C07362=1109.308,78.627,-56.858,-179.889,7.756,149.437
C07363=1109.304,78.877,-56.876,-179.889,7.759,149.437
C07364=1109.299,79.126,-56.895,-179.887,7.763,149.438
C07365=1109.295,79.375,-56.913,-179.887,7.767,149.438
C07366=1109.289,79.625,-56.931,-179.885,7.770,149.439
C07367=1109.285,79.874,-56.949,-179.885,7.774,149.440
C07368=1109.280,80.124,-56.967,-179.883,7.778,149.440
C07369=1109.275,80.372,-56.986,-179.883,7.781,149.441
C07370=1109.270,80.621,-57.004,-179.881,7.785,149.441
C07371=1109.266,80.871,-57.022,-179.880,7.790,149.442
C07372=1109.260,81.121,-57.041,-179.879,7.793,149.442
C07373=1109.255,81.370,-57.059,-179.878,7.797,149.443
C07374=1109.251,81.618,-57.078,-179.877,7.800,149.443
C07375=1109.246,81.868,-57.096,-179.876,7.804,149.444
C07376=1109.241,82.118,-57.115,-179.875,7.807,149.444
C07377=1109.236,82.367,-57.133,-179.874,7.812,149.445
C07378=1109.231,82.615,-57.151,-179.873,7.815,149.445
C07379=1109.227,82.865,-57.170,-179.872,7.819,149.446
C07380=1109.222,83.115,-57.188,-179.870,7.823,149.446
C07381=1109.217,83.363,-57.207,-179.869,7.827,149.447
C07382=1109.212,83.613,-57.225,-179.868,7.830,149.448
C07383=1109.207,83.862,-57.243,-179.867,7.834,149.448
C07384=1109.202,84.111,-57.263,-179.866,7.838,149.449
C07385=1109.198,84.361,-57.281,-179.865,7.842,149.449
C07386=1109.193,84.610,-57.299,-179.864,7.845,149.450
C07387=1109.188,84.859,-57.318,-179.863,7.849,149.450
C07388=1109.183,85.109,-57.337,-179.862,7.853,149.451
C07389=1109.179,85.358,-57.355,-179.860,7.856,149.451
C07390=1109.174,85.607,-57.373,-179.859,7.861,149.452
C07391=1109.169,85.857,-57.392,-179.858,7.864,149.452
C07392=1109.164,86.106,-57.411,-179.857,7.868,149.453
C07393=1109.159,86.355,-57.429,-179.855,7.872,149.453
C07394=1109.154,86.604,-57.448,-179.855,7.876,149.454
C07395=1109.149,86.854,-57.466,-179.853,7.879,149.454
C07396=1109.145,87.102,-57.485,-179.852,7.883,149.455
C07397=1109.140,87.352,-57.504,-179.851,7.887,149.456
C07398=1109.135,87.601,-57.523,-179.849,7.891,149.456
C07399=1109.130,87.851,-57.542,-179.848,7.895,149.456
C07400=1109.126,88.100,-57.560,-179.847,7.898,149.457
C07401=1109.121,88.349,-57.578,-179.846,7.902,149.458
C07402=1109.116,88.598,-57.598,-179.844,7.906,149.458
C07403=1109.111,88.847,-57.616,-179.844,7.909,149.459
C07404=1109.106,89.096,-57.635,-179.842,7.913,149.459
C07405=1109.101,89.346,-57.654,-179.840,7.917,149.459
C07406=1109.097,89.595,-57.672,-179.839,7.921,149.460
C07407=1109.092,89.845,-57.691,-179.838,7.925,149.461
C07408=1109.087,90.094,-57.710,-179.837,7.928,149.461
C07409=1109.082,90.343,-57.730,-179.836,7.933,149.462
C07410=1109.077,90.592,-57.748,-179.835,7.936,149.462
C07411=1109.074,90.806,-57.764,-179.833,7.940,149.462
C07412=1109.069,91.019,-57.781,-179.832,7.943,149.463
C07413=1109.065,91.234,-57.797,-179.831,7.946,149.463
C07414=1109.060,91.447,-57.813,-179.830,7.949,149.464
C07415=1109.057,91.661,-57.829,-179.829,7.953,149.464
C07416=1109.053,91.875,-57.845,-179.827,7.956,149.464
C07417=1109.049,92.088,-57.861,-179.826,7.959,149.465
C07418=1109.044,92.302,-57.878,-179.825,7.962,149.465
C07419=1109.039,92.551,-57.896,-179.824,7.966,149.466
C07420=1109.035,92.801,-57.916,-179.822,7.970,149.466
C07421=1109.030,93.050,-57.934,-179.821,7.974,149.467
C07422=1109.025,93.299,-57.954,-179.820,7.977,149.467
C07423=1109.020,93.548,-57.972,-179.818,7.981,149.468
C07424=1109.016,93.798,-57.992,-179.817,7.985,149.468
C07425=1109.011,94.046,-58.010,-179.815,7.989,149.469
C07426=1109.006,94.296,-58.030,-179.815,7.992,149.469
C07427=1109.001,94.546,-58.048,-179.813,7.996,149.470
C07428=1108.997,94.795,-58.068,-179.811,8.000,149.470
C07429=1108.991,95.044,-58.087,-179.810,8.004,149.471
C07430=1108.987,95.293,-58.106,-179.808,8.008,149.471
C07431=1108.982,95.542,-58.125,-179.807,8.012,149.471
C07432=1108.977,95.792,-58.144,-179.806,8.015,149.472
C07433=1108.972,96.041,-58.163,-179.804,8.019,149.472
C07434=1108.967,96.290,-58.182,-179.802,8.022,149.473
C07435=1108.963,96.539,-58.202,-179.801,8.026,149.473
C07436=1108.958,96.788,-58.221,-179.799,8.030,149.474
C07437=1108.953,97.038,-58.240,-179.798,8.033,149.474
C07438=1108.949,97.286,-58.259,-179.797,8.037,149.474
C07439=1108.944,97.537,-58.278,-179.795,8.041,149.475
C07440=1108.938,97.785,-58.297,-179.793,8.045,149.475
C07441=1108.934,98.035,-58.316,-179.792,8.049,149.476
C07442=1108.929,98.284,-58.336,-179.790,8.053,149.476
C07443=1108.924,98.533,-58.355,-179.789,8.057,149.477
C07444=1108.920,98.782,-58.374,-179.788,8.060,149.477
C07445=1108.915,99.031,-58.394,-179.786,8.064,149.477
C07446=1108.910,99.281,-58.413,-179.784,8.068,149.478
C07447=1108.905,99.530,-58.433,-179.783,8.071,149.478
C07448=1108.901,99.779,-58.452,-179.781,8.075,149.479
C07449=1108.896,100.028,-58.471,-179.780,8.079,149.479
C07450=1108.891,100.277,-58.491,-179.778,8.083,149.480
C07451=1108.886,100.527,-58.510,-179.776,8.087,149.480
C07452=1108.881,100.775,-58.529,-179.774,8.091,149.480
C07453=1108.877,101.025,-58.549,-179.773,8.094,149.481
C07454=1108.872,101.275,-58.568,-179.772,8.098,149.481
C07455=1108.867,101.523,-58.588,-179.770,8.101,149.482
C07456=1108.863,101.772,-58.607,-179.769,8.105,149.482
C07457=1108.858,102.022,-58.627,-179.766,8.109,149.482
C07458=1108.853,102.271,-58.646,-179.765,8.113,149.483
C07459=1108.848,102.520,-58.666,-179.763,8.117,149.483
C07460=1108.843,102.770,-58.686,-179.762,8.120,149.484
C07461=1108.839,103.018,-58.704,-179.760,8.124,149.484
C07462=1108.834,103.268,-58.724,-179.758,8.128,149.484
C07463=1108.829,103.517,-58.744,-179.756,8.132,149.485
C07464=1108.824,103.766,-58.764,-179.755,8.134,149.485
C07465=1108.819,104.015,-58.783,-179.753,8.138,149.485
C07466=1108.815,104.265,-58.803,-179.752,8.142,149.486
C07467=1108.811,104.478,-58.820,-179.750,8.146,149.486
C07468=1108.806,104.692,-58.836,-179.749,8.149,149.486
C07469=1108.802,104.905,-58.853,-179.747,8.152,149.487
C07470=1108.798,105.119,-58.870,-179.745,8.155,149.487
C07471=1108.795,105.333,-58.887,-179.744,8.158,149.487
C07472=1108.790,105.547,-58.904,-179.742,8.162,149.488
C07473=1108.786,105.760,-58.920,-179.741,8.164,149.488
C07474=1108.782,105.974,-58.938,-179.740,8.167,149.488
C07475=1108.777,106.223,-58.957,-179.738,8.171,149.488
C07476=1108.773,106.472,-58.978,-179.736,8.175,149.489
C07477=1108.768,106.722,-58.997,-179.734,8.178,149.489
C07478=1108.763,106.971,-59.017,-179.732,8.182,149.490
C07479=1108.758,107.220,-59.037,-179.730,8.186,149.490
C07480=1108.753,107.469,-59.057,-179.729,8.190,149.490
C07481=1108.749,107.719,-59.076,-179.727,8.193,149.490
C07482=1108.744,107.967,-59.096,-179.725,8.197,149.491
C07483=1108.740,108.216,-59.116,-179.723,8.201,149.491
C07484=1108.735,108.466,-59.135,-179.721,8.204,149.491
C07485=1108.730,108.715,-59.156,-179.719,8.208,149.492
C07486=1108.725,108.965,-59.176,-179.717,8.211,149.492
C07487=1108.720,109.213,-59.196,-179.716,8.215,149.492
C07488=1108.715,109.462,-59.215,-179.714,8.219,149.493
C07489=1108.711,109.711,-59.236,-179.712,8.222,149.493
C07490=1108.706,109.961,-59.255,-179.710,8.226,149.493
C07491=1108.701,110.210,-59.276,-179.708,8.230,149.494
C07492=1108.696,110.459,-59.295,-179.706,8.233,149.494
C07493=1108.692,110.708,-59.316,-179.704,8.237,149.494
C07494=1108.687,110.957,-59.335,-179.702,8.241,149.494
C07495=1108.683,111.206,-59.356,-179.700,8.244,149.495
C07496=1108.678,111.456,-59.375,-179.699,8.247,149.495
C07497=1108.673,111.704,-59.395,-179.697,8.251,149.495
C07498=1108.668,111.954,-59.415,-179.695,8.254,149.496
C07499=1108.663,112.203,-59.436,-179.693,8.258,149.496
C07500=1108.658,112.452,-59.455,-179.692,8.261,149.496
C07501=1108.654,112.701,-59.476,-179.690,8.264,149.496
C07502=1108.649,112.950,-59.496,-179.688,8.268,149.497
C07503=1108.644,113.200,-59.516,-179.686,8.272,149.497
C07504=1108.640,113.449,-59.536,-179.685,8.274,149.497
C07505=1108.635,113.697,-59.556,-179.683,8.278,149.498
C07506=1108.630,113.947,-59.577,-179.681,8.282,149.498
C07507=1108.625,114.196,-59.597,-179.680,8.284,149.498
C07508=1108.621,114.445,-59.617,-179.678,8.288,149.499
C07509=1108.616,114.694,-59.637,-179.676,8.292,149.499
C07510=1108.611,114.943,-59.657,-179.674,8.295,149.499
C07511=1108.606,115.193,-59.678,-179.673,8.298,149.500
C07512=1108.602,115.442,-59.698,-179.671,8.302,149.500
C07513=1108.597,115.691,-59.718,-179.669,8.305,149.500
C07514=1108.593,115.940,-59.739,-179.668,8.309,149.500
C07515=1108.587,116.189,-59.759,-179.666,8.312,149.501
C07516=1108.582,116.438,-59.779,-179.664,8.316,149.501
C07517=1108.578,116.687,-59.799,-179.662,8.319,149.501
C07518=1108.573,116.936,-59.820,-179.661,8.322,149.502
C07519=1108.568,117.185,-59.841,-179.659,8.326,149.502
C07520=1108.563,117.435,-59.860,-179.657,8.329,149.502
C07521=1108.559,117.684,-59.881,-179.656,8.332,149.502
C07522=1108.554,117.933,-59.901,-179.654,8.336,149.503
C07523=1108.550,118.147,-59.918,-179.652,8.338,149.503
C07524=1108.546,118.360,-59.937,-179.651,8.341,149.503
C07525=1108.542,118.574,-59.954,-179.649,8.345,149.503
C07526=1108.538,118.787,-59.971,-179.647,8.347,149.504
C07527=1108.534,119.001,-59.990,-179.646,8.350,149.504
C07528=1108.530,119.214,-60.007,-179.645,8.353,149.504
C07529=1108.526,119.428,-60.024,-179.643,8.356,149.504
C07530=1108.522,119.641,-60.042,-179.642,8.359,149.505
C07531=1108.517,119.891,-60.062,-179.640,8.362,149.505
C07532=1108.512,120.140,-60.082,-179.638,8.366,149.505
C07533=1108.508,120.389,-60.103,-179.637,8.369,149.506
C07534=1108.503,120.638,-60.124,-179.635,8.372,149.506
C07535=1108.498,120.887,-60.144,-179.633,8.376,149.506
C07536=1108.494,121.136,-60.165,-179.631,8.378,149.506
C07537=1108.489,121.385,-60.186,-179.630,8.382,149.507
C07538=1108.485,121.635,-60.206,-179.628,8.386,149.507
C07539=1108.480,121.884,-60.227,-179.625,8.389,149.507
C07540=1108.475,122.133,-60.248,-179.624,8.392,149.507
C07541=1108.471,122.382,-60.268,-179.622,8.396,149.508
C07542=1108.465,122.631,-60.289,-179.620,8.399,149.508
C07543=1108.461,122.880,-60.309,-179.619,8.402,149.508
C07544=1108.456,123.129,-60.330,-179.617,8.406,149.508
C07545=1108.451,123.378,-60.351,-179.615,8.410,149.509
C07546=1108.447,123.627,-60.372,-179.614,8.412,149.509
C07547=1108.442,123.876,-60.393,-179.612,8.416,149.509
C07548=1108.437,124.125,-60.414,-179.610,8.419,149.510
C07549=1108.433,124.374,-60.434,-179.609,8.422,149.510
C07550=1108.428,124.623,-60.454,-179.607,8.426,149.510
C07551=1108.424,124.873,-60.476,-179.605,8.429,149.511
C07552=1108.419,125.122,-60.496,-179.603,8.432,149.511
C07553=1108.414,125.371,-60.517,-179.601,8.436,149.511
C07554=1108.410,125.620,-60.538,-179.599,8.439,149.511
C07555=1108.405,125.869,-60.559,-179.598,8.442,149.512
C07556=1108.399,126.118,-60.580,-179.596,8.446,149.512
C07557=1108.395,126.367,-60.600,-179.594,8.449,149.512
C07558=1108.390,126.616,-60.621,-179.592,8.453,149.513
C07559=1108.386,126.865,-60.643,-179.591,8.456,149.513
C07560=1108.381,127.115,-60.664,-179.589,8.459,149.513
C07561=1108.377,127.364,-60.684,-179.587,8.463,149.513
C07562=1108.371,127.613,-60.705,-179.586,8.466,149.514
C07563=1108.367,127.861,-60.726,-179.584,8.469,149.514
C07564=1108.362,128.110,-60.747,-179.582,8.473,149.514
C07565=1108.357,128.360,-60.768,-179.580,8.475,149.514
C07566=1108.353,128.609,-60.789,-179.578,8.479,149.515
C07567=1108.348,128.858,-60.811,-179.576,8.483,149.515
C07568=1108.343,129.107,-60.832,-179.575,8.486,149.515
C07569=1108.339,129.356,-60.852,-179.573,8.489,149.515
C07570=1108.334,129.605,-60.874,-179.571,8.493,149.516
C07571=1108.330,129.854,-60.894,-179.570,8.496,149.516
C07572=1108.325,130.103,-60.916,-179.568,8.499,149.516
C07573=1108.320,130.352,-60.937,-179.566,8.503,149.517
C07574=1108.316,130.601,-60.957,-179.565,8.506,149.517
C07575=1108.311,130.850,-60.979,-179.563,8.509,149.517
C07576=1108.306,131.100,-61.000,-179.561,8.513,149.518
C07577=1108.301,131.349,-61.022,-179.559,8.515,149.518
C07578=1108.297,131.598,-61.043,-179.557,8.519,149.518
C07579=1108.293,131.811,-61.061,-179.556,8.522,149.518
C07580=1108.288,132.024,-61.079,-179.555,8.525,149.519
C07581=1108.284,132.239,-61.097,-179.552,8.528,149.519
C07582=1108.281,132.452,-61.115,-179.551,8.531,149.519
C07583=1108.277,132.665,-61.133,-179.550,8.534,149.519
C07584=1108.273,132.878,-61.152,-179.548,8.536,149.520
C07585=1108.268,133.092,-61.170,-179.547,8.539,149.520
C07586=1108.265,133.305,-61.189,-179.545,8.542,149.520
C07587=1108.259,133.555,-61.210,-179.544,8.546,149.520
C07588=1108.255,133.803,-61.231,-179.542,8.549,149.521
C07589=1108.251,134.053,-61.252,-179.540,8.552,149.521
C07590=1108.246,134.302,-61.274,-179.539,8.556,149.521
C07591=1108.241,134.551,-61.295,-179.536,8.559,149.522
C07592=1108.237,134.799,-61.316,-179.534,8.563,149.522
C07593=1108.232,135.049,-61.338,-179.533,8.565,149.522
C07594=1108.227,135.298,-61.359,-179.531,8.569,149.522
C07595=1108.222,135.546,-61.381,-179.529,8.573,149.523
C07596=1108.218,135.796,-61.402,-179.528,8.576,149.523
C07597=1108.214,136.045,-61.423,-179.526,8.579,149.523
C07598=1108.209,136.293,-61.445,-179.524,8.583,149.524
C07599=1108.204,136.543,-61.466,-179.523,8.586,149.524
C07600=1108.199,136.792,-61.488,-179.521,8.590,149.524
C07601=1108.194,137.041,-61.509,-179.519,8.593,149.525
C07602=1108.190,137.291,-61.531,-179.517,8.596,149.525
C07603=1108.185,137.539,-61.552,-179.515,8.599,149.525
C07604=1108.181,137.788,-61.573,-179.514,8.603,149.525
C07605=1108.176,138.038,-61.595,-179.512,8.607,149.526
C07606=1108.171,138.286,-61.616,-179.510,8.609,149.526
C07607=1108.166,138.535,-61.638,-179.509,8.613,149.526
C07608=1108.162,138.784,-61.660,-179.507,8.617,149.527
C07609=1108.157,139.033,-61.681,-179.505,8.621,149.527
C07610=1108.152,139.282,-61.703,-179.503,8.623,149.527
C07611=1108.148,139.531,-61.725,-179.501,8.627,149.527
C07612=1108.143,139.780,-61.747,-179.500,8.631,149.528
C07613=1108.139,140.029,-61.769,-179.498,8.633,149.528
C07614=1108.134,140.279,-61.790,-179.496,8.637,149.528
C07615=1108.129,140.527,-61.811,-179.495,8.641,149.529
C07616=1108.124,140.777,-61.833,-179.493,8.644,149.529
C07617=1108.120,141.025,-61.854,-179.491,8.647,149.529
C07618=1108.116,141.274,-61.876,-179.489,8.651,149.530
C07619=1108.111,141.523,-61.898,-179.487,8.654,149.530
C07620=1108.107,141.772,-61.920,-179.486,8.657,149.530
C07621=1108.102,142.022,-61.941,-179.484,8.661,149.531
C07622=1108.097,142.270,-61.963,-179.482,8.664,149.531
C07623=1108.093,142.520,-61.985,-179.481,8.668,149.531
C07624=1108.088,142.768,-62.007,-179.479,8.671,149.532
C07625=1108.083,143.017,-62.029,-179.477,8.675,149.532
C07626=1108.078,143.266,-62.051,-179.475,8.678,149.532
C07627=1108.074,143.516,-62.073,-179.474,8.682,149.533
C07628=1108.069,143.764,-62.095,-179.472,8.685,149.533
C07629=1108.064,144.014,-62.117,-179.470,8.688,149.533
C07630=1108.060,144.262,-62.138,-179.469,8.692,149.534
C07631=1108.055,144.512,-62.160,-179.467,8.696,149.534
C07632=1108.050,144.760,-62.182,-179.466,8.699,149.534
C07633=1108.046,145.010,-62.204,-179.463,8.702,149.534
C07634=1108.041,145.258,-62.226,-179.462,8.706,149.535
C07635=1108.037,145.471,-62.245,-179.460,8.709,149.535
C07636=1108.034,145.685,-62.264,-179.458,8.712,149.535
C07637=1108.029,145.899,-62.282,-179.457,8.715,149.536
C07638=1108.026,146.112,-62.302,-179.455,8.718,149.536
C07639=1108.021,146.325,-62.320,-179.453,8.721,149.536
C07640=1108.017,146.538,-62.339,-179.452,8.724,149.537
C07641=1108.013,146.752,-62.358,-179.450,8.728,149.537
C07642=1108.010,146.965,-62.376,-179.449,8.730,149.537
C07643=1108.005,147.215,-62.398,-179.447,8.734,149.537
C07644=1108.000,147.463,-62.421,-179.445,8.737,149.537
C07645=1107.996,147.712,-62.444,-179.443,8.741,149.538
C07646=1107.991,147.961,-62.465,-179.441,8.745,149.538
C07647=1107.987,148.210,-62.487,-179.439,8.748,149.538
C07648=1107.982,148.460,-62.509,-179.437,8.751,149.539
C07649=1107.977,148.708,-62.532,-179.435,8.755,149.539
C07650=1107.973,148.957,-62.554,-179.433,8.758,149.539
C07651=1107.968,149.206,-62.576,-179.431,8.761,149.539
C07652=1107.964,149.455,-62.598,-179.429,8.765,149.540
C07653=1107.958,149.704,-62.620,-179.427,8.768,149.540
C07654=1107.954,149.953,-62.643,-179.425,8.772,149.540
C07655=1107.950,150.202,-62.665,-179.423,8.776,149.540
C07656=1107.945,150.451,-62.687,-179.422,8.779,149.541
C07657=1107.940,150.700,-62.709,-179.420,8.782,149.541
C07658=1107.935,150.948,-62.732,-179.418,8.785,149.541
C07659=1107.931,151.198,-62.754,-179.416,8.789,149.541
C07660=1107.926,151.447,-62.777,-179.413,8.792,149.542
C07661=1107.921,151.695,-62.799,-179.411,8.796,149.542
C07662=1107.917,151.945,-62.821,-179.409,8.799,149.542
C07663=1107.912,152.193,-62.844,-179.407,8.802,149.542
C07664=1107.908,152.443,-62.866,-179.405,8.805,149.542
C07665=1107.903,152.692,-62.888,-179.403,8.809,149.543
C07666=1107.898,152.940,-62.911,-179.401,8.812,149.543
C07667=1107.894,153.190,-62.933,-179.399,8.816,149.543
C07668=1107.890,153.438,-62.956,-179.397,8.819,149.543
C07669=1107.884,153.687,-62.978,-179.396,8.822,149.544
C07670=1107.880,153.937,-63.000,-179.393,8.825,149.544
C07671=1107.875,154.186,-63.024,-179.391,8.829,149.544
C07672=1107.870,154.434,-63.045,-179.389,8.832,149.544
C07673=1107.866,154.683,-63.068,-179.387,8.836,149.544
C07674=1107.861,154.933,-63.091,-179.385,8.838,149.545
C07675=1107.857,155.181,-63.113,-179.383,8.842,149.545
C07676=1107.852,155.430,-63.136,-179.381,8.845,149.545
C07677=1107.848,155.679,-63.159,-179.379,8.849,149.545
C07678=1107.843,155.928,-63.180,-179.377,8.852,149.545
C07679=1107.838,156.177,-63.204,-179.375,8.854,149.546
C07680=1107.834,156.425,-63.226,-179.373,8.858,149.546
C07681=1107.829,156.675,-63.249,-179.371,8.861,149.546
C07682=1107.825,156.923,-63.271,-179.368,8.865,149.546
C07683=1107.820,157.173,-63.294,-179.366,8.868,149.546
C07684=1107.816,157.421,-63.317,-179.365,8.871,149.547
C07685=1107.811,157.670,-63.340,-179.362,8.874,149.547
C07686=1107.806,157.919,-63.362,-179.360,8.877,149.547
C07687=1107.802,158.168,-63.385,-179.358,8.881,149.547
C07688=1107.798,158.417,-63.408,-179.356,8.883,149.547
C07689=1107.793,158.667,-63.431,-179.354,8.887,149.547
C07690=1107.788,158.915,-63.453,-179.352,8.890,149.548
C07691=1107.784,159.128,-63.473,-179.350,8.892,149.548
C07692=1107.780,159.342,-63.493,-179.349,8.895,149.548
C07693=1107.776,159.554,-63.512,-179.347,8.898,149.548
C07694=1107.772,159.768,-63.532,-179.345,8.901,149.548
C07695=1107.768,159.981,-63.551,-179.343,8.903,149.548
C07696=1107.764,160.194,-63.571,-179.341,8.906,149.548
C07697=1107.761,160.408,-63.590,-179.340,8.909,149.549
C07698=1107.757,160.621,-63.610,-179.338,8.911,149.549
C07699=1107.752,160.870,-63.633,-179.336,8.915,149.549
C07700=1107.748,161.119,-63.655,-179.334,8.918,149.549
C07701=1107.743,161.368,-63.678,-179.331,8.921,149.549
C07702=1107.738,161.617,-63.702,-179.330,8.924,149.549
C07703=1107.734,161.865,-63.724,-179.327,8.927,149.549
C07704=1107.729,162.114,-63.748,-179.325,8.930,149.549
C07705=1107.724,162.364,-63.770,-179.323,8.933,149.550
C07706=1107.720,162.612,-63.793,-179.321,8.936,149.550
C07707=1107.715,162.861,-63.816,-179.319,8.939,149.550
C07708=1107.711,163.110,-63.840,-179.317,8.943,149.550
C07709=1107.706,163.358,-63.862,-179.315,8.945,149.550
C07710=1107.701,163.608,-63.885,-179.313,8.949,149.550
C07711=1107.697,163.857,-63.909,-179.310,8.952,149.551
C07712=1107.693,164.105,-63.932,-179.309,8.955,149.551
C07713=1107.688,164.354,-63.955,-179.306,8.958,149.551
C07714=1107.683,164.603,-63.978,-179.304,8.961,149.551
C07715=1107.679,164.852,-64.001,-179.302,8.964,149.551
C07716=1107.675,165.101,-64.024,-179.300,8.967,149.551
C07717=1107.670,165.350,-64.048,-179.298,8.970,149.551
C07718=1107.665,165.598,-64.071,-179.295,8.973,149.551
C07719=1107.661,165.847,-64.094,-179.294,8.976,149.552
C07720=1107.656,166.096,-64.117,-179.291,8.979,149.552
C07721=1107.651,166.345,-64.140,-179.289,8.982,149.552
C07722=1107.647,166.594,-64.164,-179.287,8.985,149.552
C07723=1107.643,166.843,-64.186,-179.285,8.988,149.552
C07724=1107.638,167.092,-64.210,-179.283,8.991,149.552
C07725=1107.633,167.341,-64.233,-179.281,8.994,149.552
C07726=1107.629,167.590,-64.256,-179.279,8.997,149.552
C07727=1107.624,167.839,-64.280,-179.276,9.000,149.553
C07728=1107.619,168.088,-64.303,-179.275,9.003,149.553
C07729=1107.615,168.337,-64.326,-179.272,9.006,149.553
C07730=1107.611,168.586,-64.349,-179.270,9.009,149.553
C07731=1107.606,168.834,-64.373,-179.268,9.012,149.553
C07732=1107.601,169.083,-64.396,-179.266,9.015,149.553
C07733=1107.596,169.332,-64.420,-179.263,9.018,149.553
C07734=1107.591,169.581,-64.443,-179.262,9.021,149.553
C07735=1107.587,169.830,-64.466,-179.259,9.024,149.553
C07736=1107.583,170.078,-64.490,-179.257,9.027,149.554
C07737=1107.578,170.327,-64.513,-179.255,9.030,149.554
C07738=1107.574,170.576,-64.537,-179.253,9.033,149.554
C07739=1107.569,170.825,-64.560,-179.251,9.036,149.554
C07740=1107.565,171.073,-64.584,-179.249,9.039,149.554
C07741=1107.560,171.322,-64.607,-179.246,9.042,149.554
C07742=1107.555,171.571,-64.631,-179.244,9.045,149.554
C07743=1107.551,171.820,-64.654,-179.242,9.048,149.554
C07744=1107.546,172.069,-64.678,-179.240,9.051,149.554
C07745=1107.541,172.318,-64.702,-179.238,9.054,149.555
C07746=1107.537,172.568,-64.725,-179.236,9.057,149.555
C07747=1107.533,172.780,-64.745,-179.234,9.059,149.555
C07748=1107.530,172.993,-64.765,-179.232,9.062,149.555
C07749=1107.526,173.206,-64.786,-179.230,9.065,149.555
C07750=1107.522,173.420,-64.806,-179.228,9.067,149.555
C07751=1107.518,173.633,-64.827,-179.226,9.069,149.555
C07752=1107.514,173.845,-64.847,-179.225,9.072,149.555
C07753=1107.510,174.059,-64.867,-179.223,9.074,149.555
C07754=1107.507,174.272,-64.887,-179.221,9.077,149.555
C07755=1107.501,174.521,-64.911,-179.219,9.080,149.556
C07756=1107.497,174.770,-64.935,-179.216,9.083,149.556
C07757=1107.492,175.019,-64.959,-179.214,9.086,149.556
C07758=1107.488,175.268,-64.982,-179.212,9.089,149.556
C07759=1107.483,175.516,-65.006,-179.210,9.092,149.556
C07760=1107.479,175.766,-65.030,-179.208,9.095,149.556
C07761=1107.475,176.014,-65.054,-179.206,9.098,149.556
C07762=1107.470,176.263,-65.077,-179.203,9.101,149.556
C07763=1107.466,176.512,-65.101,-179.201,9.104,149.556
C07764=1107.461,176.761,-65.125,-179.199,9.107,149.557
C07765=1107.456,177.009,-65.149,-179.197,9.109,149.557
C07766=1107.452,177.258,-65.172,-179.195,9.113,149.557
C07767=1107.447,177.507,-65.196,-179.192,9.116,149.557
C07768=1107.444,177.756,-65.221,-179.191,9.118,149.557
C07769=1107.438,178.005,-65.244,-179.188,9.121,149.557
C07770=1107.434,178.253,-65.269,-179.186,9.125,149.557
C07771=1107.429,178.503,-65.292,-179.184,9.127,149.557
C07772=1107.425,178.751,-65.316,-179.182,9.130,149.557
C07773=1107.420,178.999,-65.340,-179.179,9.133,149.557
C07774=1107.416,179.249,-65.364,-179.178,9.136,149.558
C07775=1107.412,179.497,-65.388,-179.175,9.139,149.558
C07776=1107.407,179.746,-65.413,-179.173,9.142,149.558
C07777=1107.402,179.995,-65.436,-179.171,9.146,149.558
C07778=1107.398,180.244,-65.460,-179.169,9.148,149.558
C07779=1107.394,180.493,-65.484,-179.166,9.151,149.558
C07780=1107.389,180.742,-65.508,-179.164,9.154,149.558
C07781=1107.384,180.991,-65.532,-179.161,9.158,149.558
C07782=1107.379,181.239,-65.556,-179.159,9.160,149.558
C07783=1107.375,181.487,-65.581,-179.157,9.163,149.558
C07784=1107.371,181.737,-65.604,-179.155,9.166,149.558
C07785=1107.366,181.986,-65.629,-179.153,9.169,149.558
C07786=1107.361,182.234,-65.653,-179.150,9.172,149.559
C07787=1107.357,182.483,-65.677,-179.148,9.175,149.559
C07788=1107.353,182.732,-65.702,-179.146,9.177,149.559
C07789=1107.348,182.981,-65.726,-179.143,9.180,149.559
C07790=1107.343,183.229,-65.750,-179.141,9.184,149.559
C07791=1107.339,183.478,-65.774,-179.138,9.187,149.559
C07792=1107.335,183.727,-65.799,-179.136,9.189,149.559
C07793=1107.330,183.976,-65.823,-179.134,9.192,149.559
C07794=1107.326,184.224,-65.847,-179.131,9.195,149.559
C07795=1107.321,184.473,-65.871,-179.130,9.198,149.559
C07796=1107.317,184.723,-65.895,-179.127,9.201,149.559
C07797=1107.312,184.971,-65.919,-179.125,9.204,149.559
C07798=1107.307,185.220,-65.944,-179.123,9.206,149.559
C07799=1107.303,185.469,-65.968,-179.120,9.210,149.559
C07800=1107.299,185.717,-65.992,-179.119,9.212,149.559
C07801=1107.294,185.966,-66.017,-179.116,9.215,149.559
C07802=1107.289,186.214,-66.041,-179.114,9.218,149.559
C07803=1107.285,186.428,-66.062,-179.112,9.220,149.559
C07804=1107.282,186.641,-66.083,-179.110,9.223,149.559
C07805=1107.277,186.854,-66.104,-179.107,9.225,149.559
C07806=1107.274,187.066,-66.125,-179.106,9.227,149.559
C07807=1107.270,187.279,-66.146,-179.104,9.229,149.559
C07808=1107.266,187.493,-66.167,-179.102,9.232,149.559
C07809=1107.262,187.706,-66.188,-179.100,9.234,149.559
C07810=1107.258,187.919,-66.209,-179.097,9.237,149.560
C07811=1107.254,188.168,-66.234,-179.095,9.240,149.560
C07812=1107.249,188.417,-66.258,-179.093,9.243,149.560
C07813=1107.245,188.666,-66.283,-179.091,9.245,149.560
C07814=1107.240,188.914,-66.307,-179.089,9.248,149.560
C07815=1107.236,189.162,-66.332,-179.086,9.251,149.560
C07816=1107.232,189.412,-66.357,-179.084,9.254,149.560
C07817=1107.227,189.660,-66.381,-179.082,9.257,149.560
C07818=1107.222,189.909,-66.406,-179.079,9.260,149.560
C07819=1107.218,190.158,-66.430,-179.077,9.262,149.560
C07820=1107.213,190.407,-66.455,-179.075,9.265,149.560
C07821=1107.209,190.656,-66.479,-179.073,9.268,149.560
C07822=1107.205,190.904,-66.505,-179.070,9.271,149.560
C07823=1107.200,191.152,-66.529,-179.068,9.274,149.560
C07824=1107.196,191.402,-66.554,-179.066,9.276,149.560
C07825=1107.191,191.650,-66.578,-179.063,9.279,149.560
C07826=1107.187,191.899,-66.604,-179.061,9.282,149.560
C07827=1107.182,192.148,-66.628,-179.059,9.285,149.560
C07828=1107.178,192.396,-66.652,-179.056,9.288,149.560
C07829=1107.173,192.646,-66.677,-179.055,9.290,149.561
C07830=1107.169,192.893,-66.702,-179.052,9.294,149.561
C07831=1107.164,193.143,-66.727,-179.050,9.297,149.561
C07832=1107.159,193.391,-66.752,-179.048,9.299,149.561
C07833=1107.156,193.640,-66.777,-179.045,9.302,149.561
C07834=1107.151,193.889,-66.802,-179.044,9.304,149.561
C07835=1107.147,194.138,-66.826,-179.041,9.308,149.561
C07836=1107.142,194.386,-66.852,-179.038,9.311,149.561
C07837=1107.137,194.635,-66.877,-179.037,9.313,149.561
C07838=1107.133,194.884,-66.901,-179.034,9.316,149.561
C07839=1107.128,195.132,-66.926,-179.032,9.320,149.561
C07840=1107.124,195.381,-66.951,-179.030,9.322,149.561
C07841=1107.120,195.629,-66.976,-179.028,9.325,149.561
C07842=1107.115,195.878,-67.001,-179.026,9.327,149.561
C07843=1107.110,196.127,-67.026,-179.023,9.330,149.561
C07844=1107.106,196.376,-67.051,-179.021,9.334,149.562
C07845=1107.102,196.625,-67.076,-179.019,9.336,149.562
C07846=1107.097,196.873,-67.101,-179.017,9.339,149.562
C07847=1107.093,197.123,-67.126,-179.014,9.343,149.562
C07848=1107.089,197.370,-67.151,-179.012,9.346,149.562
C07849=1107.084,197.620,-67.176,-179.010,9.348,149.562
C07850=1107.079,197.868,-67.201,-179.007,9.351,149.562
C07851=1107.075,198.117,-67.227,-179.005,9.354,149.562
C07852=1107.071,198.365,-67.251,-179.002,9.357,149.562
C07853=1107.066,198.614,-67.277,-179.000,9.360,149.562
C07854=1107.061,198.863,-67.302,-178.998,9.363,149.562
C07855=1107.057,199.112,-67.327,-178.995,9.366,149.562
C07856=1107.052,199.361,-67.353,-178.993,9.369,149.562
C07857=1107.048,199.609,-67.377,-178.990,9.372,149.562
C07858=1107.044,199.858,-67.403,-178.988,9.374,149.562
C07859=1107.040,200.071,-67.424,-178.985,9.377,149.562
C07860=1107.036,200.283,-67.446,-178.983,9.379,149.562
C07861=1107.032,200.496,-67.468,-178.981,9.381,149.562
C07862=1107.028,200.710,-67.489,-178.979,9.384,149.562
C07863=1107.025,200.923,-67.511,-178.976,9.387,149.562
C07864=1107.021,201.135,-67.533,-178.974,9.389,149.562
C07865=1107.017,201.348,-67.555,-178.972,9.391,149.562
C07866=1107.013,201.562,-67.576,-178.969,9.394,149.562
C07867=1107.009,201.810,-67.601,-178.968,9.396,149.562
C07868=1107.005,202.058,-67.627,-178.965,9.399,149.562
C07869=1107.000,202.306,-67.652,-178.962,9.402,149.562
C07870=1106.996,202.556,-67.677,-178.959,9.405,149.562
C07871=1106.991,202.805,-67.703,-178.956,9.408,149.562
C07872=1106.986,203.053,-67.728,-178.954,9.411,149.562
C07873=1106.982,203.302,-67.754,-178.951,9.413,149.562
C07874=1106.978,203.550,-67.780,-178.948,9.417,149.562
C07875=1106.973,203.799,-67.805,-178.945,9.419,149.561
C07876=1106.969,204.048,-67.830,-178.942,9.422,149.561
C07877=1106.964,204.297,-67.856,-178.940,9.425,149.561
C07878=1106.960,204.545,-67.881,-178.937,9.428,149.561
C07879=1106.955,204.794,-67.907,-178.934,9.431,149.561
C07880=1106.951,205.042,-67.933,-178.931,9.433,149.561
C07881=1106.946,205.291,-67.958,-178.928,9.436,149.561
C07882=1106.942,205.539,-67.984,-178.925,9.439,149.561
C07883=1106.938,205.788,-68.010,-178.923,9.442,149.561
C07884=1106.933,206.038,-68.035,-178.920,9.445,149.561
C07885=1106.929,206.286,-68.060,-178.917,9.448,149.561
C07886=1106.924,206.535,-68.086,-178.913,9.451,149.561
C07887=1106.920,206.783,-68.112,-178.911,9.454,149.560
C07888=1106.915,207.031,-68.137,-178.908,9.457,149.560
C07889=1106.911,207.280,-68.163,-178.905,9.460,149.560
C07890=1106.907,207.528,-68.189,-178.902,9.463,149.560
C07891=1106.903,207.777,-68.215,-178.899,9.465,149.560
C07892=1106.897,208.026,-68.241,-178.896,9.469,149.560
C07893=1106.893,208.274,-68.267,-178.893,9.472,149.560
C07894=1106.889,208.523,-68.293,-178.890,9.474,149.560
C07895=1106.885,208.772,-68.318,-178.887,9.478,149.560
C07896=1106.880,209.021,-68.344,-178.884,9.481,149.560
C07897=1106.876,209.269,-68.369,-178.881,9.484,149.559
C07898=1106.871,209.518,-68.395,-178.877,9.487,149.559
C07899=1106.867,209.766,-68.422,-178.875,9.490,149.559
C07900=1106.862,210.015,-68.448,-178.872,9.493,149.559
C07901=1106.858,210.264,-68.474,-178.868,9.497,149.559
C07902=1106.853,210.512,-68.499,-178.865,9.499,149.559
C07903=1106.849,210.761,-68.525,-178.862,9.503,149.559
C07904=1106.845,211.009,-68.552,-178.859,9.506,149.559
C07905=1106.840,211.258,-68.578,-178.855,9.510,149.559
C07906=1106.836,211.507,-68.603,-178.852,9.512,149.559
C07907=1106.832,211.756,-68.629,-178.849,9.516,149.559
C07908=1106.827,212.003,-68.656,-178.846,9.519,149.559
C07909=1106.822,212.252,-68.682,-178.843,9.523,149.558
C07910=1106.818,212.501,-68.707,-178.840,9.526,149.559
C07911=1106.814,212.749,-68.734,-178.837,9.529,149.558
C07912=1106.809,212.998,-68.760,-178.834,9.533,149.558
C07913=1106.805,213.247,-68.787,-178.830,9.537,149.558
C07914=1106.801,213.495,-68.812,-178.827,9.539,149.558
C07915=1106.797,213.708,-68.835,-178.826,9.542,149.558
C07916=1106.794,213.921,-68.858,-178.823,9.545,149.559
C07917=1106.790,214.134,-68.880,-178.821,9.547,149.559
C07918=1106.786,214.347,-68.902,-178.819,9.550,149.559
C07919=1106.782,214.559,-68.925,-178.817,9.552,149.559
C07920=1106.779,214.773,-68.947,-178.815,9.554,149.559
C07921=1106.774,214.985,-68.970,-178.813,9.558,149.559
C07922=1106.770,215.198,-68.992,-178.811,9.560,149.559
C07923=1106.766,215.446,-69.019,-178.809,9.563,149.559
C07924=1106.762,215.695,-69.045,-178.807,9.566,149.559
C07925=1106.758,215.943,-69.071,-178.804,9.569,149.559
C07926=1106.753,216.192,-69.098,-178.802,9.572,149.559
C07927=1106.749,216.440,-69.124,-178.799,9.575,149.559
C07928=1106.744,216.689,-69.151,-178.797,9.579,149.560
C07929=1106.740,216.938,-69.177,-178.795,9.581,149.560
C07930=1106.736,217.186,-69.203,-178.793,9.584,149.560
C07931=1106.731,217.435,-69.230,-178.790,9.587,149.560
C07932=1106.727,217.683,-69.256,-178.788,9.591,149.560
C07933=1106.722,217.932,-69.283,-178.786,9.594,149.560
C07934=1106.718,218.180,-69.309,-178.784,9.596,149.560
C07935=1106.714,218.429,-69.336,-178.781,9.599,149.560
C07936=1106.709,218.678,-69.362,-178.779,9.602,149.560
C07937=1106.705,218.926,-69.389,-178.777,9.606,149.561
C07938=1106.701,219.174,-69.415,-178.774,9.609,149.561
C07939=1106.696,219.424,-69.442,-178.772,9.612,149.561
C07940=1106.692,219.672,-69.468,-178.770,9.614,149.561
C07941=1106.687,219.920,-69.495,-178.767,9.617,149.561
C07942=1106.683,220.168,-69.522,-178.765,9.621,149.561
C07943=1106.678,220.417,-69.548,-178.763,9.624,149.561
C07944=1106.674,220.666,-69.575,-178.760,9.627,149.561
C07945=1106.670,220.915,-69.602,-178.758,9.629,149.561
C07946=1106.666,221.163,-69.628,-178.756,9.633,149.561
C07947=1106.661,221.412,-69.655,-178.754,9.636,149.562
C07948=1106.657,221.661,-69.682,-178.751,9.639,149.562
C07949=1106.653,221.909,-69.708,-178.749,9.642,149.562
C07950=1106.648,222.157,-69.735,-178.746,9.645,149.562
C07951=1106.644,222.406,-69.762,-178.744,9.648,149.562
C07952=1106.640,222.654,-69.789,-178.742,9.651,149.562
C07953=1106.635,222.903,-69.815,-178.739,9.654,149.562
C07954=1106.631,223.151,-69.842,-178.737,9.657,149.562
C07955=1106.626,223.400,-69.869,-178.734,9.660,149.562
C07956=1106.621,223.648,-69.896,-178.732,9.664,149.562
C07957=1106.618,223.897,-69.923,-178.730,9.666,149.563
C07958=1106.614,224.146,-69.950,-178.727,9.669,149.563
C07959=1106.609,224.394,-69.977,-178.725,9.672,149.563
C07960=1106.605,224.642,-70.003,-178.722,9.675,149.563
C07961=1106.600,224.891,-70.030,-178.720,9.678,149.563
C07962=1106.596,225.139,-70.057,-178.717,9.681,149.563
C07963=1106.592,225.388,-70.084,-178.716,9.684,149.563
C07964=1106.587,225.636,-70.111,-178.713,9.687,149.563
C07965=1106.583,225.885,-70.138,-178.710,9.690,149.563
C07966=1106.578,226.134,-70.165,-178.708,9.693,149.563
C07967=1106.574,226.382,-70.192,-178.705,9.696,149.563
C07968=1106.570,226.630,-70.219,-178.704,9.699,149.563
C07969=1106.565,226.879,-70.246,-178.701,9.702,149.563
C07970=1106.560,227.127,-70.273,-178.698,9.704,149.563
C07971=1106.556,227.407,-70.304,-178.696,9.708,149.563
C07972=1106.551,227.687,-70.334,-178.692,9.711,149.563
C07973=1106.546,227.967,-70.365,-178.690,9.715,149.563
C07974=1106.541,228.247,-70.395,-178.687,9.718,149.564
C07975=1106.537,228.495,-70.422,-178.684,9.720,149.563
C07976=1106.533,228.744,-70.450,-178.682,9.724,149.563
C07977=1106.528,228.992,-70.477,-178.680,9.726,149.564
C07978=1106.524,229.241,-70.504,-178.677,9.729,149.564
C07979=1106.520,229.489,-70.531,-178.674,9.732,149.563
C07980=1106.515,229.738,-70.558,-178.672,9.735,149.564
C07981=1106.511,229.986,-70.586,-178.669,9.738,149.563
C07982=1106.507,230.235,-70.613,-178.667,9.740,149.563
C07983=1106.502,230.483,-70.640,-178.665,9.743,149.564
C07984=1106.497,230.732,-70.667,-178.662,9.746,149.563
C07985=1106.494,230.980,-70.695,-178.660,9.748,149.563
C07986=1106.490,231.228,-70.722,-178.657,9.751,149.563
C07987=1106.485,231.477,-70.749,-178.654,9.754,149.563
C07988=1106.481,231.725,-70.777,-178.651,9.757,149.563
C07989=1106.477,231.974,-70.804,-178.649,9.759,149.563
C07990=1106.472,232.222,-70.831,-178.646,9.762,149.563
C07991=1106.468,232.470,-70.859,-178.644,9.765,149.563
C07992=1106.464,232.719,-70.886,-178.642,9.767,149.563
C07993=1106.459,232.968,-70.913,-178.639,9.770,149.563
C07994=1106.455,233.216,-70.941,-178.636,9.773,149.563
C07995=1106.451,233.465,-70.969,-178.633,9.776,149.563
C07996=1106.446,233.713,-70.996,-178.631,9.777,149.563
C07997=1106.442,233.961,-71.023,-178.628,9.781,149.563
C07998=1106.437,234.210,-71.050,-178.625,9.783,149.563
C07999=1106.433,234.458,-71.079,-178.623,9.785,149.563
C08000=1106.428,234.707,-71.106,-178.620,9.788,149.563
C08001=1106.425,234.956,-71.134,-178.618,9.791,149.563
C08002=1106.420,235.204,-71.161,-178.615,9.793,149.562
C08003=1106.416,235.452,-71.189,-178.612,9.796,149.562
C08004=1106.412,235.701,-71.216,-178.610,9.799,149.562
C08005=1106.407,235.949,-71.244,-178.608,9.801,149.562
C08006=1106.403,236.197,-71.271,-178.605,9.804,149.562
C08007=1106.165,225.776,-70.183,-178.710,9.689,149.563
C08008=1106.170,225.527,-70.156,-178.712,9.687,149.563
C08009=1106.173,225.278,-70.129,-178.714,9.684,149.563
C08010=1106.178,225.030,-70.102,-178.717,9.681,149.562
C08011=1106.182,224.781,-70.075,-178.719,9.678,149.562
C08012=1106.186,224.533,-70.049,-178.722,9.675,149.562
C08013=1106.191,224.285,-70.021,-178.723,9.672,149.562
C08014=1106.195,224.036,-69.994,-178.726,9.669,149.562
C08015=1106.199,223.788,-69.968,-178.729,9.666,149.562
C08016=1106.203,223.539,-69.941,-178.731,9.663,149.562
C08017=1106.208,223.290,-69.914,-178.734,9.660,149.562
C08018=1106.212,223.042,-69.888,-178.735,9.657,149.562
C08019=1106.217,222.793,-69.861,-178.738,9.654,149.562
C08020=1106.222,222.545,-69.834,-178.741,9.651,149.562
C08021=1106.226,222.296,-69.807,-178.743,9.648,149.562
C08022=1106.230,222.048,-69.780,-178.745,9.645,149.561
C08023=1106.234,221.800,-69.754,-178.748,9.642,149.561
C08024=1106.239,221.551,-69.727,-178.750,9.639,149.561
C08025=1106.244,221.302,-69.700,-178.752,9.636,149.561
C08026=1106.248,221.054,-69.674,-178.755,9.633,149.561
C08027=1106.252,220.805,-69.647,-178.757,9.629,149.561
C08028=1106.256,220.557,-69.620,-178.759,9.626,149.561
C08029=1106.261,220.307,-69.593,-178.762,9.623,149.561
C08030=1106.265,220.059,-69.566,-178.764,9.621,149.561
C08031=1106.269,219.811,-69.540,-178.766,9.618,149.561
C08032=1106.274,219.562,-69.513,-178.769,9.615,149.561
C08033=1106.278,219.313,-69.487,-178.771,9.611,149.560
C08034=1106.283,219.065,-69.460,-178.773,9.608,149.560
C08035=1106.287,218.817,-69.434,-178.775,9.606,149.560
C08036=1106.292,218.568,-69.407,-178.778,9.603,149.560
C08037=1106.296,218.319,-69.381,-178.780,9.599,149.560
C08038=1106.300,218.071,-69.354,-178.782,9.596,149.560
C08039=1106.304,217.822,-69.328,-178.785,9.593,149.560
C08040=1106.308,217.574,-69.302,-178.787,9.590,149.560
C08041=1106.313,217.325,-69.274,-178.789,9.588,149.560
C08042=1106.317,217.077,-69.249,-178.791,9.584,149.559
C08043=1106.322,216.828,-69.222,-178.794,9.581,149.559
C08044=1106.326,216.579,-69.196,-178.796,9.578,149.559
C08045=1106.331,216.331,-69.169,-178.799,9.575,149.559
C08046=1106.335,216.083,-69.142,-178.801,9.572,149.559
C08047=1106.339,215.834,-69.117,-178.803,9.569,149.559
C08048=1106.344,215.585,-69.090,-178.806,9.566,149.559
C08049=1106.348,215.337,-69.064,-178.808,9.563,149.559
C08050=1106.352,215.088,-69.037,-178.810,9.560,149.559
C08051=1106.357,214.840,-69.011,-178.812,9.557,149.559
C08052=1106.362,214.504,-68.976,-178.815,9.553,149.558
C08053=1106.369,214.169,-68.940,-178.818,9.549,149.558
C08054=1106.374,213.834,-68.904,-178.822,9.545,149.558
C08055=1106.380,213.499,-68.869,-178.825,9.541,149.558
C08056=1106.385,213.250,-68.843,-178.828,9.538,149.558
C08057=1106.389,213.001,-68.817,-178.831,9.534,149.558
C08058=1106.393,212.753,-68.791,-178.835,9.530,149.558
C08059=1106.398,212.505,-68.765,-178.837,9.527,149.558
C08060=1106.403,212.256,-68.738,-178.841,9.524,149.558
C08061=1106.407,212.007,-68.712,-178.845,9.520,149.558
C08062=1106.411,211.758,-68.687,-178.847,9.517,149.558
C08063=1106.416,211.510,-68.660,-178.851,9.514,149.558
C08064=1106.420,211.261,-68.634,-178.854,9.511,149.559
C08065=1106.424,211.012,-68.608,-178.857,9.507,149.559
C08066=1106.429,210.764,-68.583,-178.860,9.504,149.559
C08067=1106.433,210.516,-68.556,-178.863,9.501,149.559
C08068=1106.438,210.267,-68.530,-178.866,9.498,149.559
C08069=1106.442,210.018,-68.504,-178.869,9.494,149.559
C08070=1106.447,209.769,-68.478,-178.872,9.491,149.559
C08071=1106.451,209.520,-68.453,-178.876,9.488,149.559
C08072=1106.455,209.273,-68.427,-178.879,9.485,149.559
C08073=1106.460,209.024,-68.400,-178.882,9.482,149.559
C08074=1106.464,208.775,-68.374,-178.885,9.478,149.559
C08075=1106.469,208.526,-68.349,-178.888,9.476,149.559
C08076=1106.473,208.277,-68.323,-178.891,9.473,149.560
C08077=1106.478,208.029,-68.298,-178.895,9.469,149.560
C08078=1106.482,207.781,-68.272,-178.897,9.467,149.560
C08079=1106.486,207.532,-68.246,-178.900,9.464,149.560
C08080=1106.490,207.283,-68.220,-178.903,9.461,149.560
C08081=1106.496,207.035,-68.194,-178.906,9.458,149.560
C08082=1106.500,206.786,-68.169,-178.909,9.455,149.560
C08083=1106.504,206.537,-68.143,-178.912,9.452,149.560
C08084=1106.509,206.289,-68.117,-178.915,9.449,149.560
C08085=1106.513,206.040,-68.092,-178.918,9.446,149.560
C08086=1106.518,205.791,-68.066,-178.921,9.443,149.561
C08087=1106.522,205.542,-68.040,-178.924,9.440,149.561
C08088=1106.527,205.294,-68.015,-178.927,9.438,149.561
C08089=1106.531,205.046,-67.989,-178.929,9.435,149.561
C08090=1106.535,204.797,-67.963,-178.932,9.432,149.561
C08091=1106.540,204.549,-67.938,-178.935,9.429,149.561
C08092=1106.544,204.300,-67.912,-178.938,9.426,149.561
C08093=1106.548,204.051,-67.886,-178.941,9.423,149.561
C08094=1106.553,203.803,-67.861,-178.944,9.420,149.561
C08095=1106.558,203.553,-67.836,-178.946,9.417,149.561
C08096=1106.562,203.305,-67.810,-178.949,9.415,149.561
C08097=1106.567,203.057,-67.785,-178.952,9.412,149.562
C08098=1106.571,202.808,-67.759,-178.955,9.409,149.561
C08099=1106.575,202.559,-67.733,-178.957,9.406,149.562
C08100=1106.580,202.310,-67.709,-178.960,9.403,149.562
C08101=1106.585,202.061,-67.683,-178.963,9.400,149.562
C08102=1106.588,201.813,-67.658,-178.966,9.397,149.562
C08103=1106.593,201.565,-67.632,-178.968,9.394,149.562
C08104=1106.597,201.352,-67.611,-178.970,9.392,149.562
C08105=1106.600,201.138,-67.589,-178.973,9.390,149.562
C08106=1106.604,200.926,-67.567,-178.975,9.388,149.562
C08107=1106.608,200.713,-67.545,-178.977,9.385,149.562
C08108=1106.612,200.500,-67.524,-178.979,9.383,149.562
C08109=1106.616,200.286,-67.502,-178.981,9.380,149.562
C08110=1106.620,200.074,-67.480,-178.983,9.378,149.562
C08111=1106.624,199.861,-67.459,-178.986,9.375,149.562
C08112=1106.627,199.612,-67.434,-178.989,9.372,149.562
C08113=1106.632,199.364,-67.409,-178.991,9.370,149.562
C08114=1106.637,199.115,-67.384,-178.993,9.367,149.562
C08115=1106.642,198.866,-67.358,-178.996,9.364,149.562
C08116=1106.646,198.617,-67.333,-178.999,9.361,149.562
C08117=1106.650,198.369,-67.308,-179.000,9.358,149.562
C08118=1106.654,198.120,-67.283,-179.003,9.355,149.562
C08119=1106.659,197.871,-67.258,-179.005,9.352,149.562
C08120=1106.664,197.623,-67.232,-179.007,9.350,149.562
C08121=1106.668,197.374,-67.208,-179.010,9.347,149.562
C08122=1106.672,197.126,-67.182,-179.012,9.344,149.562
C08123=1106.677,196.876,-67.157,-179.015,9.341,149.562
C08124=1106.682,196.628,-67.132,-179.016,9.338,149.561
C08125=1106.686,196.379,-67.108,-179.019,9.335,149.561
C08126=1106.690,196.131,-67.082,-179.021,9.332,149.561
C08127=1106.695,195.882,-67.057,-179.023,9.329,149.561
C08128=1106.699,195.634,-67.032,-179.026,9.326,149.561
C08129=1106.704,195.384,-67.007,-179.028,9.323,149.561
C08130=1106.709,195.136,-66.983,-179.030,9.320,149.561
C08131=1106.712,194.887,-66.958,-179.032,9.317,149.561
C08132=1106.717,194.638,-66.933,-179.034,9.315,149.561
C08133=1106.721,194.390,-66.907,-179.037,9.312,149.561
C08134=1106.726,194.141,-66.883,-179.039,9.309,149.561
C08135=1106.730,193.892,-66.858,-179.041,9.306,149.561
C08136=1106.735,193.644,-66.833,-179.043,9.303,149.560
C08137=1106.739,193.394,-66.808,-179.046,9.300,149.560
C08138=1106.744,193.146,-66.783,-179.048,9.297,149.560
C08139=1106.749,192.898,-66.758,-179.050,9.294,149.560
C08140=1106.753,192.649,-66.734,-179.053,9.291,149.560
C08141=1106.758,192.400,-66.709,-179.055,9.289,149.560
C08142=1106.761,192.151,-66.684,-179.057,9.286,149.560
C08143=1106.767,191.903,-66.659,-179.059,9.284,149.560
C08144=1106.771,191.653,-66.634,-179.062,9.280,149.560
C08145=1106.775,191.405,-66.610,-179.064,9.277,149.560
C08146=1106.780,191.157,-66.585,-179.066,9.275,149.560
C08147=1106.784,190.908,-66.560,-179.069,9.272,149.560
C08148=1106.789,190.659,-66.536,-179.071,9.269,149.560
C08149=1106.793,190.410,-66.511,-179.073,9.266,149.560
C08150=1106.798,190.161,-66.486,-179.075,9.263,149.560
C08151=1106.802,189.913,-66.462,-179.077,9.261,149.560
C08152=1106.807,189.664,-66.437,-179.080,9.258,149.560
C08153=1106.811,189.415,-66.413,-179.082,9.255,149.560
C08154=1106.816,189.166,-66.388,-179.084,9.252,149.560
C08155=1106.820,188.918,-66.363,-179.087,9.249,149.560
C08156=1106.825,188.669,-66.339,-179.089,9.247,149.559
C08157=1106.829,188.420,-66.314,-179.091,9.244,149.559
C08158=1106.834,188.171,-66.290,-179.094,9.241,149.559
C08159=1106.839,187.923,-66.266,-179.096,9.238,149.559
C08160=1106.842,187.710,-66.244,-179.098,9.236,149.559
C08161=1106.846,187.497,-66.223,-179.100,9.233,149.559
C08162=1106.850,187.284,-66.202,-179.102,9.231,149.559
C08163=1106.854,187.071,-66.181,-179.104,9.228,149.559
C08164=1106.858,186.858,-66.161,-179.106,9.226,149.559
C08165=1106.862,186.644,-66.139,-179.108,9.224,149.559
C08166=1106.865,186.431,-66.119,-179.110,9.221,149.559
C08167=1106.869,186.219,-66.097,-179.111,9.219,149.559
C08168=1106.873,185.969,-66.073,-179.114,9.216,149.559
C08169=1106.879,185.720,-66.049,-179.116,9.214,149.559
C08170=1106.883,185.472,-66.025,-179.118,9.210,149.559
C08171=1106.887,185.223,-66.000,-179.121,9.207,149.559
C08172=1106.892,184.974,-65.975,-179.123,9.205,149.559
C08173=1106.896,184.726,-65.951,-179.125,9.202,149.559
C08174=1106.901,184.477,-65.927,-179.128,9.199,149.559
C08175=1106.905,184.228,-65.902,-179.130,9.196,149.559
C08176=1106.910,183.979,-65.878,-179.132,9.193,149.559
C08177=1106.915,183.731,-65.854,-179.135,9.190,149.559
C08178=1106.919,183.482,-65.829,-179.137,9.188,149.559
C08179=1106.923,183.233,-65.805,-179.139,9.185,149.558
C08180=1106.928,182.984,-65.782,-179.142,9.182,149.558
C08181=1106.933,182.735,-65.757,-179.144,9.179,149.558
C08182=1106.937,182.487,-65.733,-179.146,9.176,149.558
C08183=1106.941,182.238,-65.708,-179.148,9.173,149.558
C08184=1106.946,181.989,-65.684,-179.150,9.170,149.558
C08185=1106.951,181.740,-65.660,-179.153,9.167,149.558
C08186=1106.955,181.492,-65.636,-179.155,9.164,149.558
C08187=1106.959,181.243,-65.612,-179.157,9.162,149.558
C08188=1106.964,180.994,-65.587,-179.160,9.159,149.558
C08189=1106.969,180.745,-65.564,-179.162,9.156,149.558
C08190=1106.973,180.496,-65.540,-179.164,9.152,149.558
C08191=1106.978,180.248,-65.516,-179.166,9.150,149.558
C08192=1106.981,179.999,-65.491,-179.169,9.147,149.558
C08193=1106.987,179.750,-65.467,-179.171,9.144,149.557
C08194=1106.991,179.501,-65.443,-179.173,9.140,149.557
C08195=1106.996,179.253,-65.419,-179.175,9.138,149.557
C08196=1107.000,179.004,-65.396,-179.178,9.135,149.557
C08197=1107.004,178.755,-65.371,-179.180,9.132,149.557
C08198=1107.008,178.506,-65.347,-179.182,9.129,149.557
C08199=1107.013,178.257,-65.324,-179.184,9.126,149.557
C08200=1107.018,178.008,-65.299,-179.186,9.123,149.557
C08201=1107.023,177.759,-65.276,-179.188,9.120,149.557
C08202=1107.027,177.511,-65.252,-179.191,9.117,149.557
C08203=1107.032,177.261,-65.228,-179.192,9.114,149.556
C08204=1107.036,177.013,-65.204,-179.195,9.111,149.556
C08205=1107.040,176.764,-65.180,-179.197,9.108,149.556
C08206=1107.045,176.515,-65.157,-179.199,9.106,149.556
C08207=1107.049,176.267,-65.133,-179.201,9.102,149.556
C08208=1107.054,176.018,-65.109,-179.204,9.099,149.556
C08209=1107.058,175.770,-65.085,-179.206,9.097,149.556
C08210=1107.064,175.520,-65.061,-179.208,9.093,149.556
C08211=1107.068,175.271,-65.037,-179.210,9.090,149.556
C08212=1107.072,175.022,-65.013,-179.212,9.088,149.555
C08213=1107.077,174.774,-64.989,-179.214,9.084,149.555
C08214=1107.082,174.525,-64.966,-179.217,9.081,149.555
C08215=1107.086,174.276,-64.943,-179.219,9.079,149.555
C08216=1107.090,174.063,-64.922,-179.220,9.076,149.555
C08217=1107.093,173.850,-64.902,-179.222,9.073,149.555
C08218=1107.098,173.637,-64.882,-179.224,9.071,149.555
C08219=1107.102,173.424,-64.861,-179.226,9.068,149.555
C08220=1107.106,173.210,-64.841,-179.228,9.066,149.555
C08221=1107.109,172.997,-64.821,-179.230,9.063,149.555
C08222=1107.113,172.784,-64.801,-179.232,9.061,149.555
C08223=1107.117,172.571,-64.781,-179.233,9.058,149.554
C08224=1107.122,172.322,-64.757,-179.235,9.055,149.554
C08225=1107.126,172.074,-64.733,-179.238,9.052,149.554
C08226=1107.131,171.825,-64.710,-179.239,9.049,149.554
C08227=1107.135,171.576,-64.687,-179.242,9.046,149.554
C08228=1107.140,171.327,-64.663,-179.245,9.043,149.554
C08229=1107.144,171.078,-64.639,-179.246,9.040,149.554
C08230=1107.149,170.829,-64.616,-179.248,9.037,149.554
C08231=1107.154,170.580,-64.592,-179.251,9.034,149.554
C08232=1107.158,170.332,-64.568,-179.252,9.031,149.553
C08233=1107.163,170.083,-64.545,-179.255,9.028,149.553
C08234=1107.168,169.834,-64.522,-179.258,9.025,149.553
C08235=1107.172,169.585,-64.498,-179.259,9.022,149.553
C08236=1107.176,169.336,-64.476,-179.261,9.019,149.553
C08237=1107.181,169.088,-64.451,-179.264,9.016,149.553
C08238=1107.185,168.839,-64.428,-179.265,9.014,149.553
C08239=1107.190,168.590,-64.405,-179.268,9.010,149.553
C08240=1107.195,168.341,-64.381,-179.270,9.007,149.552
C08241=1107.199,168.092,-64.358,-179.272,9.005,149.552
C08242=1107.204,167.842,-64.335,-179.274,9.001,149.552
C08243=1107.208,167.594,-64.312,-179.277,8.998,149.552
C08244=1107.213,167.345,-64.288,-179.278,8.996,149.552
C08245=1107.217,167.096,-64.264,-179.281,8.992,149.552
C08246=1107.222,166.847,-64.241,-179.283,8.989,149.552
C08247=1107.227,166.598,-64.218,-179.285,8.986,149.552
C08248=1107.231,166.350,-64.195,-179.287,8.983,149.552
C08249=1107.235,166.101,-64.172,-179.290,8.980,149.551
C08250=1107.240,165.851,-64.148,-179.291,8.977,149.551
C08251=1107.245,165.603,-64.125,-179.294,8.974,149.551
C08252=1107.250,165.354,-64.102,-179.296,8.971,149.551
C08253=1107.254,165.105,-64.079,-179.298,8.969,149.551
C08254=1107.259,164.856,-64.056,-179.300,8.965,149.551
C08255=1107.263,164.607,-64.032,-179.302,8.962,149.551
C08256=1107.267,164.359,-64.010,-179.304,8.959,149.550
C08257=1107.272,164.110,-63.986,-179.306,8.956,149.550
C08258=1107.277,163.861,-63.963,-179.308,8.953,149.550
C08259=1107.281,163.611,-63.940,-179.310,8.950,149.550
C08260=1107.286,163.363,-63.917,-179.312,8.947,149.550
C08261=1107.291,163.114,-63.894,-179.315,8.944,149.550
C08262=1107.296,162.865,-63.871,-179.316,8.941,149.550
C08263=1107.300,162.616,-63.848,-179.319,8.938,149.550
C08264=1107.304,162.367,-63.825,-179.321,8.934,149.549
C08265=1107.308,162.118,-63.802,-179.323,8.931,149.549
C08266=1107.313,161.869,-63.779,-179.325,8.929,149.549
C08267=1107.318,161.621,-63.756,-179.327,8.925,149.549
C08268=1107.322,161.372,-63.733,-179.329,8.922,149.549
C08269=1107.327,161.123,-63.711,-179.331,8.919,149.549
C08270=1107.332,160.874,-63.687,-179.333,8.916,149.548
C08271=1107.336,160.625,-63.664,-179.335,8.913,149.548
C08272=1107.340,160.412,-63.645,-179.337,8.910,149.548
C08273=1107.344,160.198,-63.625,-179.339,8.908,149.548
C08274=1107.348,159.985,-63.605,-179.341,8.905,149.548
C08275=1107.352,159.772,-63.586,-179.343,8.902,149.548
C08276=1107.356,159.558,-63.566,-179.345,8.900,149.548
C08277=1107.360,159.346,-63.547,-179.346,8.897,149.547
C08278=1107.363,159.132,-63.528,-179.348,8.894,149.547
C08279=1107.367,158.919,-63.508,-179.349,8.892,149.547
C08280=1107.372,158.670,-63.485,-179.351,8.888,149.547
C08281=1107.377,158.421,-63.463,-179.354,8.885,149.547
C08282=1107.381,158.172,-63.439,-179.356,8.882,149.547
C08283=1107.385,157.923,-63.417,-179.358,8.879,149.546
C08284=1107.391,157.674,-63.394,-179.360,8.876,149.546
C08285=1107.395,157.426,-63.371,-179.362,8.872,149.546
C08286=1107.400,157.177,-63.348,-179.364,8.869,149.546
C08287=1107.404,156.927,-63.326,-179.366,8.866,149.546
C08288=1107.409,156.679,-63.303,-179.368,8.863,149.546
C08289=1107.414,156.430,-63.281,-179.370,8.860,149.545
C08290=1107.418,156.181,-63.258,-179.372,8.856,149.545
C08291=1107.423,155.932,-63.236,-179.374,8.853,149.545
C08292=1107.428,155.683,-63.213,-179.376,8.850,149.545
C08293=1107.432,155.434,-63.190,-179.378,8.847,149.545
C08294=1107.436,155.185,-63.168,-179.380,8.843,149.544
C08295=1107.441,154.937,-63.145,-179.383,8.840,149.544
C08296=1107.446,154.687,-63.123,-179.384,8.837,149.544
C08297=1107.450,154.438,-63.099,-179.387,8.834,149.544
C08298=1107.455,154.190,-63.078,-179.389,8.830,149.544
C08299=1107.459,153.941,-63.055,-179.391,8.827,149.543
C08300=1107.464,153.691,-63.032,-179.393,8.824,149.543
C08301=1107.469,153.443,-63.010,-179.394,8.821,149.543
C08302=1107.474,153.194,-62.987,-179.396,8.817,149.543
C08303=1107.478,152.944,-62.965,-179.398,8.814,149.543
C08304=1107.483,152.696,-62.943,-179.400,8.810,149.542
C08305=1107.488,152.446,-62.920,-179.403,8.807,149.542
C08306=1107.492,152.198,-62.897,-179.404,8.804,149.542
C08307=1107.496,151.949,-62.876,-179.407,8.801,149.542
C08308=1107.501,151.699,-62.853,-179.409,8.798,149.542
C08309=1107.506,151.451,-62.831,-179.411,8.794,149.541
C08310=1107.510,151.202,-62.809,-179.413,8.791,149.541
C08311=1107.515,150.952,-62.786,-179.415,8.787,149.541
C08312=1107.520,150.704,-62.764,-179.416,8.784,149.541
C08313=1107.524,150.455,-62.742,-179.418,8.781,149.540
C08314=1107.528,150.206,-62.720,-179.420,8.777,149.540
C08315=1107.534,149.957,-62.697,-179.422,8.774,149.540
C08316=1107.538,149.708,-62.675,-179.424,8.770,149.539
C08317=1107.543,149.459,-62.653,-179.426,8.767,149.539
C08318=1107.548,149.210,-62.630,-179.428,8.763,149.539
C08319=1107.552,148.962,-62.608,-179.430,8.760,149.539
C08320=1107.557,148.712,-62.586,-179.432,8.757,149.538
C08321=1107.561,148.463,-62.564,-179.434,8.753,149.538
C08322=1107.566,148.214,-62.541,-179.436,8.750,149.538
C08323=1107.571,147.965,-62.519,-179.438,8.746,149.538
C08324=1107.575,147.717,-62.497,-179.440,8.743,149.537
C08325=1107.580,147.467,-62.475,-179.442,8.739,149.537
C08326=1107.584,147.219,-62.453,-179.444,8.736,149.537
C08327=1107.589,146.969,-62.431,-179.446,8.732,149.536
C08328=1107.593,146.757,-62.412,-179.447,8.729,149.536
C08329=1107.597,146.542,-62.393,-179.448,8.726,149.536
C08330=1107.601,146.329,-62.375,-179.451,8.723,149.536
C08331=1107.605,146.116,-62.355,-179.452,8.720,149.535
C08332=1107.609,145.903,-62.337,-179.454,8.717,149.535
C08333=1107.613,145.690,-62.317,-179.456,8.714,149.535
C08334=1107.617,145.476,-62.299,-179.457,8.711,149.535
C08335=1107.621,145.262,-62.280,-179.459,8.708,149.535
C08336=1107.626,145.014,-62.258,-179.460,8.705,149.534
C08337=1107.630,144.765,-62.236,-179.462,8.701,149.534
C08338=1107.635,144.516,-62.214,-179.464,8.697,149.533
C08339=1107.639,144.267,-62.192,-179.466,8.694,149.533
C08340=1107.644,144.018,-62.170,-179.467,8.691,149.533
C08341=1107.648,143.769,-62.148,-179.469,8.687,149.533
C08342=1107.653,143.520,-62.126,-179.471,8.683,149.532
C08343=1107.657,143.271,-62.104,-179.473,8.680,149.532
C08344=1107.662,143.022,-62.083,-179.474,8.677,149.531
C08345=1107.667,142.772,-62.061,-179.476,8.673,149.531
C08346=1107.672,142.524,-62.040,-179.478,8.670,149.531
C08347=1107.676,142.274,-62.018,-179.479,8.666,149.530
C08348=1107.681,142.026,-61.996,-179.481,8.663,149.530
C08349=1107.685,141.776,-61.974,-179.483,8.659,149.530
C08350=1107.690,141.528,-61.952,-179.485,8.656,149.530
C08351=1107.695,141.279,-61.930,-179.487,8.652,149.529
C08352=1107.699,141.030,-61.908,-179.488,8.649,149.529
C08353=1107.704,140.781,-61.887,-179.490,8.646,149.529
C08354=1107.708,140.532,-61.865,-179.491,8.642,149.528
C08355=1107.713,140.283,-61.844,-179.493,8.638,149.528
C08356=1107.718,140.033,-61.822,-179.495,8.636,149.528
C08357=1107.723,139.785,-61.800,-179.497,8.632,149.527
C08358=1107.728,139.536,-61.778,-179.499,8.628,149.527
C08359=1107.732,139.287,-61.756,-179.500,8.626,149.527
C08360=1107.737,139.037,-61.735,-179.502,8.622,149.526
C08361=1107.742,138.789,-61.714,-179.504,8.618,149.526
C08362=1107.746,138.539,-61.692,-179.506,8.615,149.526
C08363=1107.751,138.291,-61.670,-179.507,8.612,149.526
C08364=1107.755,138.041,-61.648,-179.509,8.608,149.525
C08365=1107.760,137.792,-61.627,-179.511,8.605,149.525
C08366=1107.765,137.544,-61.606,-179.512,8.602,149.525
C08367=1107.769,137.295,-61.584,-179.514,8.598,149.524
C08368=1107.774,137.045,-61.563,-179.516,8.595,149.524
C08369=1107.779,136.797,-61.541,-179.518,8.591,149.524
C08370=1107.783,136.547,-61.519,-179.519,8.588,149.523
C08371=1107.788,136.298,-61.498,-179.521,8.585,149.523
C08372=1107.793,136.049,-61.476,-179.523,8.581,149.523
C08373=1107.797,135.800,-61.455,-179.524,8.578,149.523
C08374=1107.802,135.551,-61.434,-179.526,8.574,149.522
C08375=1107.807,135.302,-61.412,-179.529,8.571,149.522
C08376=1107.811,135.053,-61.390,-179.530,8.568,149.522
C08377=1107.816,134.804,-61.369,-179.532,8.564,149.521
C08378=1107.820,134.556,-61.348,-179.534,8.561,149.521
C08379=1107.825,134.306,-61.327,-179.535,8.557,149.521
C08380=1107.830,134.057,-61.305,-179.537,8.554,149.521
C08381=1107.835,133.808,-61.284,-179.539,8.551,149.520
C08382=1107.840,133.559,-61.263,-179.541,8.547,149.520
C08383=1107.843,133.310,-61.241,-179.542,8.544,149.520
C08384=1107.848,133.096,-61.223,-179.543,8.541,149.519
C08385=1107.852,132.883,-61.205,-179.545,8.538,149.519
C08386=1107.856,132.670,-61.187,-179.547,8.535,149.519
C08387=1107.860,132.456,-61.169,-179.548,8.533,149.519
C08388=1107.863,132.243,-61.150,-179.550,8.530,149.518
C08389=1107.868,132.029,-61.131,-179.551,8.527,149.518
C08390=1107.872,131.816,-61.113,-179.553,8.524,149.518
C08391=1107.876,131.602,-61.096,-179.555,8.521,149.518
C08392=1107.881,131.353,-61.074,-179.556,8.518,149.517
C08393=1107.885,131.104,-61.054,-179.558,8.514,149.517
C08394=1107.890,130.855,-61.032,-179.560,8.511,149.517
C08395=1107.895,130.606,-61.011,-179.561,8.508,149.517
C08396=1107.899,130.358,-60.990,-179.563,8.504,149.516
C08397=1107.904,130.108,-60.968,-179.565,8.501,149.516
C08398=1107.909,129.858,-60.947,-179.566,8.498,149.516
C08399=1107.913,129.610,-60.926,-179.568,8.495,149.516
C08400=1107.918,129.361,-60.905,-179.570,8.491,149.515
C08401=1107.923,129.112,-60.884,-179.572,8.488,149.515
C08402=1107.928,128.863,-60.863,-179.574,8.484,149.515
C08403=1107.932,128.613,-60.842,-179.576,8.481,149.514
C08404=1107.937,128.364,-60.821,-179.577,8.478,149.514
C08405=1107.941,128.116,-60.800,-179.579,8.474,149.514
C08406=1107.947,127.866,-60.779,-179.581,8.471,149.513
C08407=1107.951,127.617,-60.759,-179.583,8.467,149.513
C08408=1107.956,127.368,-60.738,-179.584,8.464,149.513
C08409=1107.961,127.119,-60.716,-179.586,8.461,149.513
C08410=1107.965,126.870,-60.695,-179.588,8.457,149.512
C08411=1107.970,126.621,-60.674,-179.589,8.455,149.512
C08412=1107.975,126.372,-60.654,-179.591,8.451,149.512
C08413=1107.979,126.123,-60.632,-179.593,8.447,149.511
C08414=1107.984,125.874,-60.612,-179.595,8.444,149.511
C08415=1107.989,125.625,-60.591,-179.597,8.441,149.511
C08416=1107.993,125.375,-60.570,-179.598,8.437,149.511
C08417=1107.998,125.126,-60.549,-179.600,8.434,149.510
C08418=1108.002,124.878,-60.528,-179.602,8.431,149.510
C08419=1108.007,124.628,-60.507,-179.604,8.427,149.510
C08420=1108.012,124.379,-60.487,-179.605,8.424,149.509
C08421=1108.017,124.130,-60.466,-179.607,8.421,149.509
C08422=1108.021,123.881,-60.445,-179.609,8.417,149.509
C08423=1108.027,123.632,-60.424,-179.610,8.415,149.509
C08424=1108.031,123.383,-60.404,-179.612,8.411,149.508
C08425=1108.036,123.133,-60.383,-179.614,8.407,149.508
C08426=1108.040,122.884,-60.362,-179.616,8.405,149.508
C08427=1108.045,122.635,-60.341,-179.618,8.401,149.508
C08428=1108.049,122.386,-60.320,-179.619,8.397,149.507
C08429=1108.054,122.138,-60.300,-179.621,8.394,149.507
C08430=1108.059,121.888,-60.279,-179.623,8.391,149.507
C08431=1108.063,121.639,-60.259,-179.625,8.387,149.507
C08432=1108.069,121.390,-60.238,-179.626,8.384,149.506
C08433=1108.073,121.141,-60.217,-179.628,8.381,149.506
C08434=1108.077,120.892,-60.197,-179.630,8.377,149.506
C08435=1108.083,120.643,-60.176,-179.632,8.374,149.505
C08436=1108.087,120.394,-60.156,-179.633,8.371,149.505
C08437=1108.092,120.145,-60.135,-179.635,8.367,149.505
C08438=1108.097,119.896,-60.114,-179.637,8.364,149.504
C08439=1108.101,119.646,-60.095,-179.639,8.361,149.504
C08440=1108.105,119.433,-60.076,-179.640,8.357,149.504
C08441=1108.110,119.219,-60.059,-179.642,8.354,149.504
C08442=1108.114,119.005,-60.042,-179.643,8.352,149.503
C08443=1108.118,118.792,-60.024,-179.644,8.349,149.503
C08444=1108.122,118.578,-60.006,-179.646,8.346,149.503
C08445=1108.126,118.365,-59.989,-179.647,8.344,149.503
C08446=1108.130,118.152,-59.971,-179.649,8.340,149.502
C08447=1108.134,117.938,-59.954,-179.651,8.337,149.502
C08448=1108.138,117.689,-59.933,-179.652,8.334,149.502
C08449=1108.143,117.440,-59.912,-179.654,8.331,149.502
C08450=1108.148,117.190,-59.893,-179.656,8.327,149.501
C08451=1108.153,116.941,-59.872,-179.657,8.325,149.501
C08452=1108.157,116.692,-59.852,-179.659,8.321,149.501
C08453=1108.162,116.443,-59.831,-179.661,8.317,149.500
C08454=1108.167,116.194,-59.811,-179.663,8.314,149.500
C08455=1108.171,115.945,-59.791,-179.664,8.311,149.500
C08456=1108.176,115.696,-59.771,-179.666,8.307,149.500
C08457=1108.181,115.446,-59.750,-179.668,8.304,149.499
C08458=1108.185,115.197,-59.729,-179.669,8.300,149.499
C08459=1108.190,114.948,-59.710,-179.671,8.297,149.499
C08460=1108.195,114.700,-59.690,-179.673,8.293,149.498
C08461=1108.200,114.450,-59.669,-179.674,8.290,149.498
C08462=1108.205,114.201,-59.649,-179.676,8.287,149.498
C08463=1108.210,113.952,-59.629,-179.678,8.283,149.498
C08464=1108.214,113.703,-59.608,-179.680,8.279,149.497
C08465=1108.219,113.453,-59.589,-179.681,8.277,149.497
C08466=1108.224,113.204,-59.568,-179.684,8.273,149.497
C08467=1108.228,112.955,-59.547,-179.685,8.269,149.496
C08468=1108.233,112.706,-59.528,-179.687,8.266,149.496
C08469=1108.238,112.457,-59.508,-179.689,8.263,149.496
C08470=1108.243,112.208,-59.487,-179.690,8.259,149.495
C08471=1108.247,111.959,-59.468,-179.692,8.256,149.495
C08472=1108.252,111.710,-59.447,-179.693,8.253,149.495
C08473=1108.257,111.460,-59.427,-179.695,8.249,149.494
C08474=1108.262,111.211,-59.407,-179.697,8.246,149.494
C08475=1108.266,110.961,-59.387,-179.699,8.242,149.494
C08476=1108.271,110.713,-59.367,-179.701,8.238,149.494
C08477=1108.276,110.464,-59.347,-179.703,8.235,149.493
C08478=1108.281,110.215,-59.327,-179.705,8.231,149.493
C08479=1108.285,109.965,-59.307,-179.707,8.227,149.493
C08480=1108.290,109.716,-59.287,-179.709,8.224,149.492
C08481=1108.295,109.467,-59.268,-179.711,8.220,149.492
C08482=1108.300,109.218,-59.247,-179.713,8.216,149.492
C08483=1108.304,108.969,-59.228,-179.715,8.213,149.492
C08484=1108.309,108.720,-59.207,-179.716,8.210,149.491
C08485=1108.313,108.470,-59.188,-179.718,8.206,149.491
C08486=1108.319,108.222,-59.168,-179.720,8.203,149.491
C08487=1108.323,107.972,-59.148,-179.721,8.199,149.490
C08488=1108.328,107.723,-59.128,-179.723,8.195,149.490
C08489=1108.332,107.474,-59.108,-179.725,8.192,149.490
C08490=1108.337,107.224,-59.088,-179.727,8.188,149.489
C08491=1108.342,106.976,-59.068,-179.729,8.184,149.489
C08492=1108.347,106.727,-59.049,-179.731,8.181,149.489
C08493=1108.352,106.477,-59.029,-179.732,8.177,149.488
C08494=1108.356,106.228,-59.008,-179.734,8.173,149.488
C08495=1108.362,105.979,-58.989,-179.736,8.169,149.488
C08496=1108.365,105.766,-58.972,-179.737,8.167,149.487
C08497=1108.370,105.551,-58.956,-179.739,8.163,149.487
C08498=1108.374,105.338,-58.938,-179.740,8.160,149.487
C08499=1108.377,105.124,-58.921,-179.742,8.157,149.486
C08500=1108.382,104.911,-58.904,-179.743,8.154,149.486
C08501=1108.386,104.697,-58.888,-179.745,8.151,149.486
C08502=1108.390,104.483,-58.871,-179.747,8.147,149.486
C08503=1108.394,104.270,-58.854,-179.748,8.144,149.485
C08504=1108.399,104.020,-58.834,-179.750,8.141,149.485
C08505=1108.404,103.771,-58.815,-179.752,8.137,149.485
C08506=1108.408,103.522,-58.795,-179.753,8.133,149.484
C08507=1108.413,103.273,-58.775,-179.755,8.129,149.484
C08508=1108.418,103.024,-58.756,-179.757,8.126,149.483
C08509=1108.422,102.775,-58.737,-179.758,8.122,149.483
C08510=1108.427,102.525,-58.717,-179.759,8.119,149.483
C08511=1108.432,102.276,-58.698,-179.761,8.115,149.482
C08512=1108.437,102.027,-58.678,-179.763,8.111,149.482
C08513=1108.442,101.778,-58.658,-179.765,8.107,149.481
C08514=1108.446,101.529,-58.639,-179.766,8.103,149.481
C08515=1108.451,101.279,-58.619,-179.768,8.099,149.481
C08516=1108.456,101.030,-58.600,-179.770,8.096,149.480
C08517=1108.461,100.781,-58.580,-179.772,8.092,149.480
C08518=1108.465,100.532,-58.561,-179.773,8.089,149.479
C08519=1108.470,100.283,-58.542,-179.774,8.085,149.479
C08520=1108.475,100.033,-58.522,-179.776,8.081,149.479
C08521=1108.480,99.784,-58.503,-179.777,8.077,149.478
C08522=1108.485,99.535,-58.484,-179.779,8.073,149.478
C08523=1108.489,99.286,-58.464,-179.781,8.070,149.477
C08524=1108.495,99.037,-58.445,-179.783,8.066,149.477
C08525=1108.499,98.787,-58.426,-179.784,8.062,149.477
C08526=1108.503,98.538,-58.406,-179.785,8.059,149.476
C08527=1108.509,98.289,-58.387,-179.787,8.055,149.476
C08528=1108.513,98.039,-58.368,-179.788,8.051,149.475
C08529=1108.518,97.791,-58.349,-179.790,8.047,149.475
C08530=1108.523,97.541,-58.329,-179.792,8.044,149.474
C08531=1108.528,97.292,-58.310,-179.793,8.040,149.474
C08532=1108.532,97.043,-58.291,-179.794,8.037,149.474
C08533=1108.537,96.794,-58.271,-179.796,8.033,149.473
C08534=1108.542,96.545,-58.252,-179.797,8.029,149.473
C08535=1108.547,96.295,-58.234,-179.799,8.025,149.472
C08536=1108.552,96.046,-58.214,-179.801,8.021,149.472
C08537=1108.557,95.796,-58.195,-179.802,8.017,149.471
C08538=1108.561,95.548,-58.176,-179.803,8.014,149.471
C08539=1108.566,95.298,-58.156,-179.804,8.010,149.470
C08540=1108.571,95.050,-58.138,-179.806,8.006,149.470
C08541=1108.576,94.800,-58.119,-179.807,8.002,149.469
C08542=1108.581,94.551,-58.099,-179.809,7.998,149.469
C08543=1108.585,94.302,-58.080,-179.810,7.995,149.469
C08544=1108.590,94.052,-58.061,-179.812,7.991,149.468
C08545=1108.594,93.803,-58.042,-179.813,7.987,149.468
C08546=1108.599,93.553,-58.023,-179.814,7.983,149.467
C08547=1108.604,93.305,-58.004,-179.816,7.979,149.467
C08548=1108.609,93.056,-57.985,-179.817,7.976,149.466
C08549=1108.614,92.806,-57.965,-179.819,7.972,149.466
C08550=1108.619,92.557,-57.947,-179.820,7.968,149.465
C08551=1108.624,92.307,-57.928,-179.821,7.964,149.465
C08552=1108.628,92.093,-57.912,-179.823,7.961,149.464
C08553=1108.632,91.880,-57.896,-179.824,7.958,149.464
C08554=1108.635,91.667,-57.879,-179.825,7.955,149.464
C08555=1108.640,91.453,-57.863,-179.826,7.952,149.463
C08556=1108.644,91.239,-57.847,-179.827,7.948,149.463
C08557=1108.648,91.025,-57.830,-179.828,7.945,149.462
C08558=1108.653,90.811,-57.815,-179.829,7.942,149.462
C08559=1108.656,90.598,-57.798,-179.830,7.939,149.461
C08560=1108.662,90.348,-57.779,-179.832,7.935,149.461
C08561=1108.666,90.099,-57.760,-179.833,7.931,149.461
C08562=1108.671,89.850,-57.742,-179.834,7.927,149.460
C08563=1108.676,89.600,-57.723,-179.835,7.923,149.459
C08564=1108.680,89.352,-57.704,-179.837,7.920,149.459
C08565=1108.686,89.102,-57.685,-179.838,7.915,149.458
C08566=1108.690,88.853,-57.666,-179.839,7.912,149.458
C08567=1108.695,88.603,-57.648,-179.841,7.908,149.458
C08568=1108.699,88.354,-57.629,-179.842,7.904,149.457
C08569=1108.704,88.105,-57.611,-179.843,7.901,149.456
C08570=1108.710,87.856,-57.591,-179.844,7.897,149.456
C08571=1108.714,87.606,-57.573,-179.846,7.893,149.455
C08572=1108.719,87.357,-57.554,-179.847,7.890,149.455
C08573=1108.724,87.108,-57.535,-179.848,7.885,149.454
C08574=1108.728,86.859,-57.517,-179.849,7.881,149.454
C08575=1108.734,86.610,-57.498,-179.850,7.878,149.453
C08576=1108.738,86.360,-57.479,-179.851,7.874,149.453
C08577=1108.743,86.111,-57.461,-179.853,7.870,149.452
C08578=1108.748,85.862,-57.442,-179.854,7.867,149.452
C08579=1108.752,85.612,-57.424,-179.855,7.863,149.451
C08580=1108.757,85.364,-57.405,-179.857,7.859,149.451
C08581=1108.763,85.114,-57.386,-179.857,7.855,149.450
C08582=1108.767,84.864,-57.368,-179.859,7.851,149.450
C08583=1108.772,84.616,-57.349,-179.860,7.847,149.449
C08584=1108.777,84.366,-57.331,-179.861,7.844,149.449
C08585=1108.781,84.117,-57.312,-179.862,7.840,149.448
C08586=1108.786,83.868,-57.294,-179.863,7.837,149.448
C08587=1108.792,83.618,-57.275,-179.865,7.833,149.447
C08588=1108.796,83.369,-57.256,-179.866,7.829,149.446
C08589=1108.801,83.120,-57.238,-179.867,7.825,149.446
C08590=1108.806,82.871,-57.220,-179.868,7.821,149.445
C08591=1108.810,82.621,-57.200,-179.869,7.818,149.445
C08592=1108.815,82.372,-57.182,-179.870,7.814,149.444
C08593=1108.820,82.123,-57.164,-179.871,7.811,149.444
C08594=1108.825,81.874,-57.146,-179.872,7.806,149.443
C08595=1108.830,81.624,-57.127,-179.874,7.802,149.443
C08596=1108.835,81.375,-57.109,-179.874,7.799,149.442
C08597=1108.840,81.126,-57.091,-179.876,7.795,149.442
C08598=1108.844,80.877,-57.072,-179.876,7.792,149.441
C08599=1108.849,80.627,-57.054,-179.877,7.787,149.440
C08600=1108.854,80.378,-57.035,-179.878,7.784,149.440
C08601=1108.859,80.129,-57.017,-179.879,7.780,149.439
C08602=1108.864,79.879,-56.999,-179.880,7.777,149.439
C08603=1108.868,79.630,-56.980,-179.881,7.772,149.438
C08604=1108.873,79.381,-56.962,-179.882,7.769,149.438
C08605=1108.879,79.132,-56.944,-179.884,7.765,149.437
C08606=1108.883,78.882,-56.925,-179.884,7.762,149.437
C08607=1108.888,78.633,-56.907,-179.886,7.758,149.436
C08608=1108.892,78.419,-56.892,-179.887,7.755,149.436
C08609=1108.896,78.205,-56.875,-179.888,7.751,149.435
C08610=1108.901,77.992,-56.860,-179.888,7.748,149.435
C08611=1108.904,77.777,-56.845,-179.889,7.745,149.434
C08612=1108.908,77.564,-56.829,-179.890,7.742,149.434
C08613=1108.913,77.351,-56.813,-179.891,7.739,149.433
C08614=1108.917,77.136,-56.798,-179.891,7.736,149.433
C08615=1108.921,76.922,-56.782,-179.892,7.733,149.432
C08616=1108.926,76.673,-56.764,-179.893,7.729,149.432
C08617=1108.931,76.423,-56.746,-179.895,7.725,149.431
C08618=1108.936,76.174,-56.728,-179.896,7.721,149.431
C08619=1108.940,75.925,-56.710,-179.898,7.717,149.430
C08620=1108.945,75.676,-56.692,-179.899,7.713,149.430
C08621=1108.951,75.426,-56.673,-179.901,7.709,149.429
C08622=1108.955,75.177,-56.654,-179.902,7.705,149.429
C08623=1108.960,74.928,-56.636,-179.903,7.701,149.428
C08624=1108.965,74.679,-56.618,-179.905,7.697,149.428
C08625=1108.970,74.430,-56.600,-179.907,7.693,149.427
C08626=1108.975,74.180,-56.583,-179.908,7.689,149.427
C08627=1108.980,73.931,-56.565,-179.909,7.686,149.426
C08628=1108.984,73.681,-56.547,-179.910,7.682,149.426
C08629=1108.989,73.432,-56.529,-179.911,7.677,149.425
C08630=1108.994,73.182,-56.511,-179.913,7.674,149.425
C08631=1108.999,72.933,-56.493,-179.915,7.670,149.424
C08632=1109.004,72.684,-56.475,-179.916,7.666,149.424
C08633=1109.009,72.435,-56.457,-179.917,7.661,149.423
C08634=1109.014,72.186,-56.439,-179.919,7.658,149.423
C08635=1109.019,71.936,-56.421,-179.920,7.654,149.422
C08636=1109.023,71.687,-56.403,-179.921,7.649,149.422
C08637=1109.028,71.437,-56.385,-179.922,7.646,149.421
C08638=1109.032,71.188,-56.368,-179.924,7.642,149.421
C08639=1109.037,70.939,-56.350,-179.925,7.638,149.420
C08640=1109.042,70.690,-56.332,-179.927,7.634,149.420
C08641=1109.047,70.440,-56.314,-179.928,7.630,149.419
C08642=1109.052,70.191,-56.296,-179.929,7.626,149.419
C08643=1109.057,69.941,-56.279,-179.931,7.622,149.418
C08644=1109.062,69.692,-56.261,-179.933,7.618,149.418
C08645=1109.067,69.443,-56.243,-179.933,7.615,149.417
C08646=1109.072,69.194,-56.225,-179.935,7.611,149.417
C08647=1109.077,68.945,-56.207,-179.936,7.607,149.416
C08648=1109.081,68.695,-56.190,-179.937,7.603,149.416
C08649=1109.086,68.446,-56.172,-179.939,7.599,149.415
C08650=1109.091,68.197,-56.154,-179.940,7.595,149.415
C08651=1109.096,67.947,-56.137,-179.942,7.591,149.414
C08652=1109.101,67.698,-56.119,-179.943,7.587,149.414
C08653=1109.106,67.449,-56.101,-179.944,7.583,149.413
C08654=1109.110,67.200,-56.084,-179.945,7.579,149.413
C08655=1109.115,66.950,-56.066,-179.947,7.575,149.412
C08656=1109.120,66.701,-56.048,-179.948,7.571,149.412
C08657=1109.125,66.452,-56.030,-179.949,7.567,149.411
C08658=1109.131,66.202,-56.013,-179.951,7.563,149.411
C08659=1109.135,65.953,-55.996,-179.952,7.559,149.410
C08660=1109.140,65.703,-55.979,-179.953,7.556,149.410
C08661=1109.145,65.454,-55.961,-179.954,7.551,149.409
C08662=1109.150,65.205,-55.943,-179.956,7.548,149.409
C08663=1109.154,64.955,-55.926,-179.957,7.544,149.408
C08664=1109.158,64.741,-55.911,-179.958,7.541,149.408
C08665=1109.163,64.527,-55.895,-179.960,7.537,149.407
C08666=1109.167,64.314,-55.880,-179.960,7.533,149.407
C08667=1109.171,64.100,-55.865,-179.961,7.530,149.406
C08668=1109.175,63.885,-55.851,-179.963,7.526,149.406
C08669=1109.180,63.671,-55.836,-179.964,7.523,149.405
C08670=1109.183,63.458,-55.820,-179.965,7.520,149.405
C08671=1109.188,63.244,-55.805,-179.966,7.517,149.404
C08672=1109.193,62.994,-55.788,-179.967,7.513,149.404
C08673=1109.197,62.745,-55.771,-179.968,7.509,149.403
C08674=1109.203,62.496,-55.753,-179.970,7.505,149.403
C08675=1109.208,62.246,-55.736,-179.971,7.500,149.402
C08676=1109.212,61.997,-55.719,-179.972,7.496,149.402
C08677=1109.217,61.748,-55.701,-179.973,7.493,149.401
C08678=1109.222,61.498,-55.684,-179.975,7.489,149.401
C08679=1109.226,61.249,-55.666,-179.976,7.485,149.400
C08680=1109.232,60.999,-55.649,-179.977,7.481,149.400
C08681=1109.237,60.750,-55.632,-179.979,7.477,149.399
C08682=1109.241,60.501,-55.614,-179.980,7.473,149.399
C08683=1109.247,60.252,-55.597,-179.981,7.470,149.398
C08684=1109.251,60.003,-55.580,-179.982,7.465,149.397
C08685=1109.256,59.753,-55.563,-179.983,7.461,149.397
C08686=1109.261,59.503,-55.545,-179.985,7.457,149.396
C08687=1109.266,59.254,-55.528,-179.986,7.453,149.396
C08688=1109.271,59.004,-55.511,-179.987,7.449,149.395
C08689=1109.275,58.755,-55.494,-179.988,7.446,149.395
C08690=1109.281,58.507,-55.477,-179.989,7.441,149.394
C08691=1109.286,58.257,-55.459,-179.991,7.438,149.394
C08692=1109.290,58.007,-55.443,-179.992,7.433,149.393
C08693=1109.296,57.757,-55.425,-179.993,7.429,149.393
C08694=1109.300,57.509,-55.408,-179.994,7.426,149.392
C08695=1109.305,57.259,-55.391,-179.995,7.422,149.392
C08696=1109.310,57.010,-55.374,-179.997,7.418,149.391
C08697=1109.315,56.760,-55.357,-179.998,7.414,149.391
C08698=1109.320,56.511,-55.340,-179.999,7.409,149.390
C08699=1109.325,56.262,-55.322,179.999,7.405,149.389
C08700=1109.329,56.012,-55.306,179.999,7.402,149.389
C08701=1109.335,55.763,-55.289,179.998,7.398,149.388
C08702=1109.339,55.514,-55.272,179.996,7.394,149.388
C08703=1109.344,55.264,-55.254,179.995,7.389,149.387
C08704=1109.349,55.015,-55.238,179.993,7.386,149.387
C08705=1109.354,54.765,-55.220,179.993,7.382,149.386
C08706=1109.359,54.516,-55.204,179.991,7.378,149.386
C08707=1109.364,54.266,-55.187,179.990,7.374,149.385
C08708=1109.369,54.017,-55.170,179.989,7.370,149.384
C08709=1109.374,53.768,-55.152,179.988,7.366,149.384
C08710=1109.379,53.519,-55.136,179.987,7.362,149.383
C08711=1109.383,53.270,-55.119,179.986,7.358,149.383
C08712=1109.389,53.020,-55.102,179.985,7.354,149.382
C08713=1109.393,52.770,-55.085,179.983,7.350,149.381
C08714=1109.399,52.521,-55.068,179.982,7.346,149.381
C08715=1109.403,52.272,-55.052,179.981,7.342,149.380
C08716=1109.408,52.022,-55.035,179.980,7.338,149.380
C08717=1109.414,51.773,-55.018,179.979,7.334,149.379
C08718=1109.418,51.524,-55.001,179.978,7.330,149.379
C08719=1109.423,51.274,-54.984,179.976,7.326,149.378
C08720=1109.427,51.060,-54.970,179.976,7.322,149.377
C08721=1109.431,50.846,-54.955,179.975,7.319,149.377
C08722=1109.436,50.632,-54.942,179.974,7.316,149.377
C08723=1109.440,50.418,-54.927,179.972,7.312,149.376
C08724=1109.444,50.204,-54.912,179.972,7.309,149.376
C08725=1109.449,49.990,-54.898,179.971,7.305,149.375
C08726=1109.453,49.776,-54.884,179.970,7.302,149.375
C08727=1109.457,49.562,-54.869,179.969,7.298,149.374
C08728=1109.462,49.313,-54.852,179.968,7.295,149.374
C08729=1109.466,49.063,-54.836,179.967,7.291,149.373
C08730=1109.472,48.814,-54.820,179.966,7.286,149.372
C08731=1109.477,48.564,-54.803,179.964,7.282,149.372
C08732=1109.481,48.315,-54.786,179.963,7.278,149.371
C08733=1109.486,48.066,-54.770,179.963,7.275,149.371
C08734=1109.491,47.816,-54.753,179.961,7.271,149.370
C08735=1109.496,47.567,-54.736,179.960,7.266,149.369
C08736=1109.501,47.318,-54.720,179.959,7.262,149.369
C08737=1109.506,47.068,-54.703,179.958,7.259,149.368
C08738=1109.511,46.818,-54.687,179.957,7.255,149.368
C08739=1109.516,46.569,-54.670,179.956,7.250,149.367
C08740=1109.521,46.320,-54.653,179.955,7.246,149.366
C08741=1109.525,46.070,-54.637,179.954,7.242,149.366
C08742=1109.530,45.821,-54.620,179.953,7.239,149.365
C08743=1109.536,45.572,-54.603,179.952,7.234,149.365
C08744=1109.541,45.322,-54.588,179.951,7.230,149.364
C08745=1109.545,45.073,-54.571,179.950,7.226,149.363
C08746=1109.550,44.823,-54.554,179.948,7.222,149.363
C08747=1109.555,44.574,-54.538,179.948,7.218,149.362
C08748=1109.560,44.324,-54.522,179.946,7.214,149.362
C08749=1109.566,44.075,-54.505,179.945,7.210,149.361
C08750=1109.570,43.826,-54.488,179.944,7.205,149.360
C08751=1109.575,43.576,-54.472,179.943,7.202,149.360
C08752=1109.580,43.327,-54.456,179.942,7.198,149.359
C08753=1109.584,43.077,-54.440,179.941,7.194,149.359
C08754=1109.590,42.829,-54.423,179.940,7.189,149.358
C08755=1109.595,42.578,-54.407,179.940,7.186,149.357
C08756=1109.600,42.329,-54.390,179.939,7.182,149.357
C08757=1109.605,42.079,-54.374,179.937,7.178,149.356
C08758=1109.610,41.831,-54.358,179.936,7.173,149.356
C08759=1109.615,41.581,-54.341,179.935,7.169,149.355
C08760=1109.620,41.332,-54.326,179.934,7.166,149.354
C08761=1109.624,41.082,-54.309,179.933,7.161,149.354
C08762=1109.629,40.833,-54.292,179.932,7.157,149.353
C08763=1109.634,40.583,-54.277,179.931,7.153,149.352
C08764=1109.639,40.334,-54.260,179.931,7.149,149.352
C08765=1109.644,40.084,-54.245,179.929,7.145,149.351
C08766=1109.649,39.835,-54.228,179.928,7.141,149.350
C08767=1109.654,39.586,-54.212,179.927,7.137,149.350
C08768=1109.659,39.336,-54.195,179.926,7.132,149.349
C08769=1109.665,39.086,-54.180,179.926,7.129,149.349
C08770=1109.669,38.837,-54.163,179.924,7.124,149.348
C08771=1109.674,38.587,-54.147,179.923,7.120,149.347
C08772=1109.680,38.339,-54.131,179.922,7.116,149.347
C08773=1109.684,38.089,-54.115,179.922,7.112,149.346
C08774=1109.689,37.840,-54.099,179.921,7.108,149.345
C08775=1109.694,37.590,-54.083,179.920,7.104,149.345
C08776=1109.698,37.376,-54.068,179.919,7.101,149.344
C08777=1109.702,37.162,-54.055,179.918,7.097,149.344
C08778=1109.707,36.947,-54.041,179.917,7.093,149.343
C08779=1109.711,36.734,-54.028,179.916,7.090,149.342
C08780=1109.715,36.520,-54.014,179.916,7.086,149.342
C08781=1109.719,36.306,-54.000,179.915,7.083,149.341
C08782=1109.723,36.092,-53.986,179.914,7.079,149.341
C08783=1109.728,35.877,-53.973,179.913,7.076,149.340
C08784=1109.733,35.628,-53.957,179.912,7.071,149.340
C08785=1109.738,35.378,-53.940,179.912,7.068,149.339
C08786=1109.743,35.129,-53.925,179.910,7.063,149.338
C08787=1109.748,34.879,-53.909,179.909,7.059,149.338
C08788=1109.753,34.630,-53.893,179.908,7.055,149.337
C08789=1109.758,34.381,-53.877,179.908,7.051,149.336
C08790=1109.763,34.131,-53.861,179.907,7.047,149.335
C08791=1109.768,33.882,-53.845,179.906,7.042,149.335
C08792=1109.772,33.632,-53.829,179.905,7.038,149.334
C08793=1109.778,33.383,-53.814,179.904,7.034,149.333
C08794=1109.783,33.134,-53.797,179.904,7.030,149.333
C08795=1109.787,32.884,-53.781,179.903,7.026,149.332
C08796=1109.793,32.634,-53.766,179.902,7.022,149.331
C08797=1109.798,32.386,-53.750,179.900,7.017,149.331
C08798=1109.803,32.135,-53.734,179.900,7.014,149.330
C08799=1109.807,31.886,-53.719,179.899,7.009,149.330
C08800=1109.812,31.636,-53.703,179.898,7.005,149.329
C08801=1109.817,31.388,-53.686,179.897,7.000,149.328
C08802=1109.823,31.138,-53.671,179.897,6.997,149.327
C08803=1109.827,30.888,-53.655,179.896,6.993,149.327
C08804=1109.833,30.639,-53.639,179.895,6.988,149.326
C08805=1109.837,30.390,-53.624,179.894,6.984,149.325
C08806=1109.842,30.140,-53.608,179.893,6.980,149.325
C08807=1109.847,29.891,-53.592,179.893,6.976,149.324
C08808=1109.853,29.641,-53.576,179.892,6.971,149.323
C08809=1109.857,29.391,-53.561,179.891,6.967,149.323
C08810=1109.862,29.142,-53.545,179.890,6.963,149.322
C08811=1109.868,28.893,-53.530,179.889,6.959,149.321
C08812=1109.872,28.643,-53.514,179.888,6.955,149.320
C08813=1109.877,28.394,-53.498,179.887,6.950,149.320
C08814=1109.882,28.145,-53.483,179.886,6.946,149.319
C08815=1109.887,27.895,-53.467,179.886,6.942,149.318
C08816=1109.892,27.645,-53.451,179.885,6.938,149.317
C08817=1109.897,27.396,-53.436,179.884,6.933,149.317
C08818=1109.902,27.147,-53.421,179.883,6.929,149.316
C08819=1109.907,26.897,-53.405,179.882,6.925,149.316
C08820=1109.912,26.647,-53.390,179.882,6.921,149.315
C08821=1109.917,26.398,-53.374,179.881,6.917,149.314
C08822=1109.922,26.149,-53.358,179.880,6.912,149.313
C08823=1109.927,25.899,-53.343,179.880,6.908,149.312
C08824=1109.932,25.649,-53.327,179.879,6.904,149.312
C08825=1109.937,25.400,-53.312,179.878,6.900,149.311
C08826=1109.942,25.151,-53.297,179.877,6.895,149.310
C08827=1109.947,24.901,-53.281,179.876,6.891,149.310
C08828=1109.952,24.651,-53.265,179.875,6.886,149.309
C08829=1109.957,24.402,-53.250,179.875,6.882,149.308
C08830=1109.962,24.153,-53.235,179.874,6.878,149.307
C08831=1109.968,23.904,-53.219,179.873,6.874,149.307
C08832=1109.971,23.690,-53.206,179.873,6.870,149.306
C08833=1109.976,23.475,-53.193,179.872,6.867,149.305
C08834=1109.980,23.260,-53.179,179.871,6.862,149.305
C08835=1109.984,23.047,-53.167,179.871,6.859,149.304
C08836=1109.988,22.833,-53.153,179.871,6.855,149.303
C08837=1109.993,22.618,-53.140,179.870,6.852,149.303
C08838=1109.997,22.404,-53.127,179.869,6.848,149.302
C08839=1110.001,22.190,-53.113,179.869,6.844,149.301
C08840=1110.006,21.941,-53.098,179.868,6.840,149.301
C08841=1110.011,21.690,-53.083,179.868,6.836,149.300
C08842=1110.016,21.441,-53.068,179.867,6.832,149.299
C08843=1110.021,21.192,-53.053,179.866,6.827,149.299
C08844=1110.027,20.942,-53.037,179.865,6.823,149.298
C08845=1110.031,20.693,-53.022,179.864,6.818,149.297
C08846=1110.037,20.444,-53.006,179.864,6.814,149.296
C08847=1110.041,20.193,-52.992,179.863,6.810,149.296
C08848=1110.046,19.944,-52.976,179.862,6.805,149.295
C08849=1110.051,19.695,-52.961,179.861,6.801,149.294
C08850=1110.056,19.446,-52.946,179.861,6.797,149.293
C08851=1110.061,19.196,-52.931,179.860,6.793,149.292
C08852=1110.067,18.946,-52.916,179.860,6.788,149.292
C08853=1110.071,18.697,-52.901,179.859,6.784,149.291
C08854=1110.076,18.447,-52.885,179.858,6.779,149.290
C08855=1110.081,18.198,-52.871,179.858,6.775,149.289
C08856=1110.087,17.948,-52.855,179.857,6.771,149.289
C08857=1110.091,17.699,-52.840,179.857,6.766,149.288
C08858=1110.097,17.450,-52.824,179.856,6.762,149.287
C08859=1110.102,17.200,-52.810,179.855,6.757,149.286
C08860=1110.106,16.951,-52.795,179.855,6.753,149.285
C08861=1110.112,16.701,-52.780,179.854,6.749,149.285
C08862=1110.117,16.452,-52.765,179.853,6.744,149.284
C08863=1110.122,16.202,-52.750,179.852,6.740,149.283
C08864=1110.126,15.953,-52.734,179.852,6.735,149.282
C08865=1110.132,15.703,-52.719,179.852,6.731,149.281
C08866=1110.136,15.453,-52.704,179.851,6.727,149.281
C08867=1110.141,15.204,-52.690,179.850,6.722,149.280
C08868=1110.147,14.954,-52.675,179.850,6.717,149.279
C08869=1110.151,14.705,-52.660,179.849,6.713,149.278
C08870=1110.156,14.456,-52.645,179.849,6.709,149.277
C08871=1110.162,14.206,-52.630,179.848,6.705,149.276
C08872=1110.167,13.956,-52.615,179.848,6.700,149.275
C08873=1110.172,13.707,-52.600,179.847,6.696,149.275
C08874=1110.177,13.457,-52.586,179.846,6.691,149.274
C08875=1110.182,13.208,-52.571,179.846,6.687,149.273
C08876=1110.187,12.959,-52.555,179.846,6.682,149.272
C08877=1110.192,12.709,-52.541,179.845,6.678,149.272
C08878=1110.197,12.460,-52.526,179.844,6.673,149.271
C08879=1110.202,12.210,-52.511,179.843,6.668,149.270
C08880=1110.207,11.961,-52.496,179.843,6.664,149.269
C08881=1110.212,11.711,-52.482,179.842,6.660,149.268
C08882=1110.217,11.462,-52.467,179.842,6.656,149.267
C08883=1110.222,11.212,-52.452,179.841,6.651,149.266
C08884=1110.227,10.963,-52.437,179.841,6.646,149.266
C08885=1110.232,10.713,-52.422,179.840,6.641,149.265
C08886=1110.238,10.463,-52.408,179.840,6.637,149.264
C08887=1110.242,10.214,-52.393,179.839,6.633,149.263
C08888=1110.246,9.999,-52.380,179.839,6.628,149.262
C08889=1110.251,9.785,-52.368,179.838,6.625,149.262
C08890=1110.255,9.571,-52.354,179.838,6.621,149.261
C08891=1110.259,9.357,-52.342,179.838,6.617,149.260
C08892=1110.264,9.142,-52.329,179.837,6.613,149.259
C08893=1110.268,8.928,-52.317,179.837,6.610,149.259
C08894=1110.272,8.714,-52.304,179.837,6.606,149.258
C08895=1110.276,8.499,-52.291,179.836,6.601,149.257
C08896=1110.281,8.250,-52.277,179.835,6.597,149.256
C08897=1110.286,8.000,-52.263,179.834,6.592,149.255
C08898=1110.291,7.751,-52.248,179.835,6.588,149.254
C08899=1110.297,7.501,-52.233,179.834,6.583,149.254
C08900=1110.302,7.252,-52.219,179.833,6.579,149.253
C08901=1110.307,7.003,-52.204,179.832,6.574,149.252
C08902=1110.312,6.753,-52.190,179.832,6.570,149.251
C08903=1110.317,6.503,-52.175,179.831,6.565,149.250
C08904=1110.321,6.254,-52.160,179.831,6.560,149.249
C08905=1110.327,6.004,-52.146,179.830,6.556,149.249
C08906=1110.332,5.755,-52.131,179.829,6.551,149.248
C08907=1110.337,5.505,-52.117,179.829,6.546,149.247
C08908=1110.342,5.256,-52.102,179.828,6.542,149.246
C08909=1110.347,5.006,-52.088,179.827,6.537,149.245
C08910=1110.352,4.756,-52.073,179.827,6.533,149.245
C08911=1110.357,4.507,-52.060,179.826,6.528,149.244
C08912=1110.363,4.258,-52.044,179.826,6.523,149.243
C08913=1110.368,4.008,-52.030,179.825,6.519,149.242
C08914=1110.373,3.759,-52.015,179.824,6.514,149.241
C08915=1110.377,3.509,-52.001,179.823,6.509,149.240
C08916=1110.382,3.259,-51.987,179.823,6.505,149.239
C08917=1110.387,3.009,-51.973,179.823,6.501,149.239
C08918=1110.392,2.760,-51.958,179.822,6.497,149.238
C08919=1110.398,2.511,-51.944,179.821,6.492,149.237
C08920=1110.403,2.262,-51.929,179.821,6.487,149.236
C08921=1110.407,2.012,-51.915,179.820,6.483,149.235
C08922=1110.412,1.762,-51.901,179.819,6.478,149.235
C08923=1110.417,1.512,-51.887,179.819,6.473,149.234
C08924=1110.422,1.263,-51.872,179.818,6.469,149.233
C08925=1110.428,1.014,-51.858,179.817,6.464,149.232
C08926=1110.433,0.764,-51.844,179.817,6.460,149.231
C08927=1110.438,0.515,-51.829,179.816,6.455,149.230
C08928=1110.442,0.265,-51.815,179.816,6.450,149.229
C08929=1110.447,0.016,-51.801,179.815,6.447,149.229
C08930=1110.453,-0.233,-51.787,179.815,6.442,149.228
C08931=1110.458,-0.483,-51.772,179.814,6.437,149.227
C08932=1110.463,-0.733,-51.758,179.813,6.433,149.226
C08933=1110.468,-0.983,-51.744,179.813,6.428,149.225
C08934=1110.473,-1.232,-51.730,179.812,6.423,149.225
C08935=1110.478,-1.481,-51.716,179.812,6.419,149.224
C08936=1110.483,-1.731,-51.701,179.811,6.414,149.223
C08937=1110.488,-1.981,-51.687,179.810,6.410,149.222
C08938=1110.493,-2.230,-51.673,179.810,6.405,149.221
C08939=1110.499,-2.479,-51.659,179.809,6.401,149.221
C08940=1110.504,-2.730,-51.645,179.809,6.397,149.220
C08941=1110.509,-2.980,-51.631,179.808,6.392,149.219
C08942=1110.514,-3.229,-51.617,179.808,6.387,149.218
C08943=1110.520,-3.478,-51.603,179.807,6.383,149.217
C08944=1110.523,-3.693,-51.590,179.806,6.379,149.217
C08945=1110.528,-3.907,-51.578,179.806,6.375,149.216
C08946=1110.532,-4.121,-51.566,179.805,6.371,149.215
C08947=1110.536,-4.336,-51.555,179.805,6.368,149.214
C08948=1110.541,-4.550,-51.543,179.804,6.363,149.214
C08949=1110.545,-4.765,-51.530,179.804,6.360,149.213
C08950=1110.549,-4.978,-51.518,179.804,6.356,149.212
C08951=1110.554,-5.193,-51.507,179.803,6.351,149.211
C08952=1110.559,-5.443,-51.493,179.802,6.347,149.211
C08953=1110.564,-5.692,-51.478,179.801,6.342,149.210
C08954=1110.569,-5.942,-51.464,179.801,6.338,149.209
C08955=1110.574,-6.191,-51.451,179.801,6.334,149.208
C08956=1110.579,-6.441,-51.437,179.800,6.329,149.207
C08957=1110.584,-6.691,-51.423,179.799,6.325,149.207
C08958=1110.589,-6.940,-51.409,179.799,6.320,149.206
C08959=1110.594,-7.190,-51.395,179.798,6.316,149.205
C08960=1110.600,-7.440,-51.381,179.797,6.311,149.204
C08961=1110.605,-7.689,-51.368,179.797,6.306,149.203
C08962=1110.609,-7.938,-51.354,179.796,6.302,149.202
C08963=1110.614,-8.188,-51.339,179.796,6.298,149.202
C08964=1110.620,-8.438,-51.326,179.795,6.293,149.201
C08965=1110.624,-8.687,-51.312,179.795,6.289,149.200
C08966=1110.629,-8.937,-51.298,179.794,6.284,149.199
C08967=1110.635,-9.186,-51.284,179.793,6.279,149.198
C08968=1110.640,-9.436,-51.271,179.793,6.275,149.197
C08969=1110.645,-9.685,-51.257,179.792,6.270,149.196
C08970=1110.650,-9.935,-51.243,179.791,6.266,149.196
C08971=1110.655,-10.185,-51.230,179.791,6.261,149.195
C08972=1110.661,-10.434,-51.216,179.791,6.257,149.194
C08973=1110.665,-10.683,-51.202,179.790,6.252,149.193
C08974=1110.670,-10.934,-51.188,179.789,6.248,149.192
C08975=1110.676,-11.183,-51.174,179.789,6.243,149.192
C08976=1110.680,-11.433,-51.162,179.788,6.239,149.191
C08977=1110.686,-11.682,-51.148,179.788,6.234,149.190
C08978=1110.691,-11.931,-51.133,179.787,6.229,149.189
C08979=1110.695,-12.181,-51.120,179.786,6.225,149.188
C08980=1110.701,-12.430,-51.106,179.786,6.220,149.187
C08981=1110.706,-12.681,-51.093,179.786,6.216,149.186
C08982=1110.711,-12.929,-51.080,179.786,6.211,149.186
C08983=1110.716,-13.180,-51.066,179.785,6.207,149.185
C08984=1110.722,-13.429,-51.052,179.784,6.202,149.184
C08985=1110.726,-13.678,-51.038,179.784,6.198,149.183
C08986=1110.731,-13.929,-51.025,179.783,6.193,149.182
C08987=1110.736,-14.177,-51.012,179.783,6.188,149.181
C08988=1110.741,-14.428,-50.998,179.782,6.184,149.181
C08989=1110.747,-14.677,-50.984,179.781,6.179,149.180
C08990=1110.752,-14.927,-50.971,179.781,6.174,149.179
C08991=1110.757,-15.176,-50.957,179.781,6.170,149.178
C08992=1110.762,-15.426,-50.944,179.780,6.166,149.177
C08993=1110.767,-15.675,-50.931,179.780,6.161,149.176
C08994=1110.772,-15.925,-50.917,179.779,6.157,149.175
C08995=1110.778,-16.174,-50.904,179.778,6.152,149.175
C08996=1110.783,-16.424,-50.890,179.778,6.147,149.174
C08997=1110.788,-16.673,-50.877,179.777,6.142,149.173
C08998=1110.793,-16.923,-50.863,179.777,6.138,149.172
C08999=1110.798,-17.172,-50.850,179.776,6.133,149.171
C09000=1110.802,-17.388,-50.839,179.776,6.129,149.170
C09001=1110.806,-17.601,-50.827,179.775,6.125,149.170
C09002=1110.811,-17.816,-50.815,179.775,6.121,149.169
C09003=1110.816,-18.031,-50.804,179.775,6.118,149.168
C09004=1110.819,-18.246,-50.793,179.774,6.113,149.167
C09005=1110.824,-18.459,-50.781,179.774,6.109,149.166
C09006=1110.829,-18.674,-50.770,179.774,6.106,149.166
C09007=1110.833,-18.889,-50.758,179.773,6.101,149.165
C09008=1110.838,-19.138,-50.745,179.772,6.097,149.164
C09009=1110.843,-19.388,-50.731,179.772,6.092,149.163
C09010=1110.848,-19.638,-50.718,179.771,6.087,149.162
C09011=1110.854,-19.887,-50.705,179.771,6.083,149.162
C09012=1110.859,-20.136,-50.692,179.771,6.079,149.161
C09013=1110.863,-20.386,-50.679,179.770,6.074,149.160
C09014=1110.869,-20.636,-50.666,179.770,6.069,149.159
C09015=1110.873,-20.885,-50.652,179.769,6.064,149.158
C09016=1110.879,-21.135,-50.639,179.769,6.060,149.157
C09017=1110.884,-21.385,-50.626,179.768,6.055,149.156
C09018=1110.889,-21.634,-50.613,179.768,6.050,149.155
C09019=1110.895,-21.884,-50.600,179.767,6.046,149.154
C09020=1110.900,-22.133,-50.586,179.767,6.041,149.153
C09021=1110.905,-22.383,-50.573,179.766,6.036,149.153
C09022=1110.909,-22.633,-50.560,179.766,6.031,149.152
C09023=1110.915,-22.882,-50.547,179.765,6.027,149.151
C09024=1110.920,-23.132,-50.534,179.765,6.022,149.150
C09025=1110.925,-23.381,-50.520,179.764,6.017,149.149
C09026=1110.930,-23.631,-50.508,179.764,6.012,149.148
C09027=1110.935,-23.880,-50.495,179.764,6.008,149.147
C09028=1110.941,-24.130,-50.481,179.763,6.003,149.146
C09029=1110.946,-24.380,-50.469,179.763,5.998,149.145
C09030=1110.950,-24.630,-50.456,179.763,5.993,149.144
C09031=1110.956,-24.879,-50.443,179.762,5.988,149.143
C09032=1110.961,-25.128,-50.429,179.762,5.984,149.142
C09033=1110.965,-25.378,-50.416,179.761,5.979,149.141
C09034=1110.971,-25.628,-50.403,179.761,5.974,149.141
C09035=1110.976,-25.877,-50.391,179.761,5.970,149.140
C09036=1110.981,-26.127,-50.378,179.761,5.965,149.139
C09037=1110.987,-26.377,-50.364,179.761,5.961,149.138
C09038=1110.992,-26.626,-50.352,179.762,5.957,149.136
C09039=1110.996,-26.876,-50.339,179.761,5.952,149.136
C09040=1111.002,-27.125,-50.326,179.762,5.948,149.134
C09041=1111.007,-27.375,-50.313,179.761,5.943,149.134
C09042=1111.012,-27.625,-50.300,179.761,5.939,149.133
C09043=1111.017,-27.874,-50.288,179.762,5.935,149.132
C09044=1111.023,-28.124,-50.274,179.762,5.930,149.131
C09045=1111.027,-28.374,-50.261,179.762,5.926,149.130
C09046=1111.033,-28.623,-50.249,179.762,5.921,149.129
C09047=1111.038,-28.872,-50.236,179.762,5.917,149.128
C09048=1111.043,-29.123,-50.223,179.761,5.912,149.127
C09049=1111.048,-29.372,-50.210,179.761,5.909,149.126
C09050=1111.053,-29.621,-50.197,179.762,5.905,149.125
C09051=1111.058,-29.871,-50.185,179.761,5.900,149.124
C09052=1111.063,-30.121,-50.172,179.761,5.896,149.123
C09053=1111.069,-30.370,-50.159,179.761,5.891,149.122
C09054=1111.074,-30.620,-50.146,179.761,5.886,149.121
C09055=1111.078,-30.870,-50.133,179.761,5.882,149.120
C09056=1111.083,-31.084,-50.122,179.761,5.879,149.119
C09057=1111.088,-31.299,-50.112,179.760,5.875,149.119
C09058=1111.092,-31.514,-50.100,179.760,5.871,149.118
C09059=1111.096,-31.728,-50.090,179.760,5.868,149.117
C09060=1111.101,-31.942,-50.078,179.760,5.864,149.116
C09061=1111.105,-32.157,-50.068,179.759,5.859,149.116
C09062=1111.110,-32.371,-50.056,179.759,5.856,149.115
C09063=1111.114,-32.585,-50.046,179.759,5.852,149.114
C09064=1111.119,-32.835,-50.034,179.759,5.847,149.113
C09065=1111.124,-33.085,-50.021,179.759,5.843,149.112
C09066=1111.130,-33.335,-50.008,179.758,5.838,149.111
C09067=1111.135,-33.584,-49.995,179.757,5.834,149.111
C09068=1111.140,-33.834,-49.982,179.758,5.830,149.110
C09069=1111.145,-34.084,-49.969,179.757,5.825,149.109
C09070=1111.150,-34.334,-49.958,179.757,5.821,149.108
C09071=1111.155,-34.583,-49.945,179.756,5.816,149.107
C09072=1111.160,-34.832,-49.932,179.756,5.812,149.106
C09073=1111.165,-35.082,-49.920,179.755,5.808,149.105
C09074=1111.171,-35.333,-49.907,179.755,5.803,149.105
C09075=1111.176,-35.582,-49.894,179.755,5.798,149.104
C09076=1111.181,-35.831,-49.882,179.754,5.793,149.103
C09077=1111.186,-36.081,-49.869,179.754,5.789,149.102
C09078=1111.192,-36.330,-49.857,179.753,5.784,149.101
C09079=1111.196,-36.580,-49.844,179.752,5.780,149.100
C09080=1111.201,-36.830,-49.832,179.752,5.776,149.099
C09081=1111.206,-37.079,-49.819,179.752,5.771,149.098
C09082=1111.212,-37.329,-49.807,179.751,5.766,149.097
C09083=1111.217,-37.578,-49.795,179.751,5.761,149.097
C09084=1111.222,-37.828,-49.782,179.750,5.756,149.096
C09085=1111.228,-38.078,-49.770,179.749,5.751,149.095
C09086=1111.232,-38.328,-49.757,179.749,5.747,149.094
C09087=1111.237,-38.577,-49.744,179.748,5.742,149.093
C09088=1111.243,-38.827,-49.733,179.748,5.737,149.092
C09089=1111.248,-39.076,-49.720,179.747,5.733,149.091
C09090=1111.253,-39.326,-49.707,179.746,5.728,149.091
C09091=1111.258,-39.575,-49.696,179.746,5.723,149.090
C09092=1111.263,-39.825,-49.683,179.745,5.718,149.089
C09093=1111.269,-40.075,-49.671,179.744,5.713,149.088
C09094=1111.273,-40.325,-49.658,179.744,5.708,149.087
C09095=1111.279,-40.575,-49.646,179.743,5.703,149.086
C09096=1111.284,-40.824,-49.634,179.743,5.698,149.085
C09097=1111.289,-41.073,-49.621,179.742,5.693,149.084
C09098=1111.294,-41.323,-49.609,179.741,5.688,149.083
C09099=1111.300,-41.573,-49.596,179.741,5.683,149.083
C09100=1111.305,-41.823,-49.585,179.740,5.678,149.082
C09101=1111.310,-42.072,-49.572,179.739,5.673,149.081
C09102=1111.316,-42.322,-49.560,179.739,5.668,149.080
C09103=1111.321,-42.571,-49.548,179.738,5.663,149.079
C09104=1111.326,-42.821,-49.536,179.737,5.657,149.078
C09105=1111.331,-43.070,-49.524,179.737,5.653,149.077
C09106=1111.336,-43.320,-49.512,179.737,5.648,149.076
C09107=1111.340,-43.570,-49.499,179.738,5.644,149.075
C09108=1111.346,-43.820,-49.487,179.738,5.638,149.074
C09109=1111.351,-44.070,-49.475,179.738,5.633,149.072
C09110=1111.356,-44.319,-49.462,179.738,5.629,149.072
C09111=1111.362,-44.569,-49.451,179.738,5.624,149.070
C09112=1111.366,-44.783,-49.440,179.738,5.620,149.070
C09113=1111.370,-44.998,-49.430,179.738,5.616,149.069
C09114=1111.375,-45.212,-49.420,179.738,5.612,149.068
C09115=1111.380,-45.427,-49.409,179.739,5.608,149.067
C09116=1111.384,-45.642,-49.399,179.739,5.605,149.066
C09117=1111.388,-45.856,-49.388,179.738,5.600,149.065
C09118=1111.393,-46.071,-49.378,179.739,5.595,149.064
C09119=1111.397,-46.286,-49.368,179.739,5.592,149.063
C09120=1111.402,-46.535,-49.355,179.739,5.588,149.062
C09121=1111.408,-46.785,-49.344,179.739,5.582,149.061
C09122=1111.413,-47.035,-49.332,179.739,5.577,149.060
C09123=1111.418,-47.284,-49.319,179.740,5.573,149.059
C09124=1111.423,-47.534,-49.308,179.740,5.568,149.058
C09125=1111.428,-47.784,-49.296,179.740,5.564,149.056
C09126=1111.433,-48.033,-49.283,179.740,5.559,149.055
C09127=1111.439,-48.283,-49.271,179.740,5.554,149.054
C09128=1111.444,-48.533,-49.260,179.741,5.550,149.053
C09129=1111.449,-48.783,-49.248,179.741,5.545,149.052
C09130=1111.454,-49.032,-49.236,179.740,5.540,149.051
C09131=1111.459,-49.282,-49.224,179.741,5.536,149.050
C09132=1111.465,-49.532,-49.212,179.741,5.530,149.049
C09133=1111.469,-49.781,-49.200,179.742,5.526,149.048
C09134=1111.475,-50.031,-49.188,179.741,5.521,149.047
C09135=1111.481,-50.280,-49.177,179.741,5.516,149.046
C09136=1111.485,-50.530,-49.165,179.742,5.512,149.044
C09137=1111.491,-50.779,-49.153,179.742,5.507,149.044
C09138=1111.496,-51.029,-49.141,179.742,5.502,149.042
C09139=1111.501,-51.279,-49.129,179.742,5.498,149.041
C09140=1111.506,-51.528,-49.118,179.742,5.493,149.040
C09141=1111.512,-51.778,-49.106,179.743,5.489,149.039
C09142=1111.517,-52.028,-49.093,179.743,5.483,149.038
C09143=1111.521,-52.277,-49.082,179.742,5.479,149.037
C09144=1111.527,-52.527,-49.070,179.743,5.474,149.036
C09145=1111.532,-52.777,-49.058,179.743,5.469,149.035
C09146=1111.537,-53.027,-49.047,179.743,5.464,149.034
C09147=1111.542,-53.277,-49.035,179.743,5.460,149.033
C09148=1111.548,-53.525,-49.023,179.743,5.455,149.032
C09149=1111.553,-53.775,-49.011,179.744,5.451,149.031
C09150=1111.558,-54.025,-48.999,179.744,5.446,149.030
C09151=1111.564,-54.275,-48.988,179.744,5.441,149.028
C09152=1111.568,-54.525,-48.976,179.744,5.437,149.027
C09153=1111.574,-54.774,-48.964,179.744,5.432,149.026
C09154=1111.579,-55.024,-48.952,179.744,5.427,149.025
C09155=1111.584,-55.274,-48.941,179.744,5.423,149.024
C09156=1111.589,-55.524,-48.929,179.744,5.418,149.023
C09157=1111.594,-55.772,-48.918,179.745,5.413,149.022
C09158=1111.600,-56.022,-48.906,179.745,5.408,149.021
C09159=1111.604,-56.272,-48.894,179.745,5.403,149.020
C09160=1111.610,-56.522,-48.883,179.745,5.399,149.019
C09161=1111.615,-56.772,-48.871,179.745,5.394,149.018
C09162=1111.620,-57.021,-48.859,179.745,5.389,149.017
C09163=1111.625,-57.271,-48.848,179.745,5.385,149.016
C09164=1111.631,-57.520,-48.837,179.746,5.380,149.015
C09165=1111.636,-57.770,-48.825,179.746,5.375,149.013
C09166=1111.641,-58.020,-48.813,179.746,5.371,149.012
C09167=1111.646,-58.270,-48.802,179.746,5.366,149.011
C09168=1111.651,-58.485,-48.792,179.746,5.362,149.010
C09169=1111.655,-58.699,-48.782,179.746,5.358,149.009
C09170=1111.660,-58.914,-48.772,179.746,5.354,149.009
C09171=1111.664,-59.128,-48.762,179.747,5.350,149.008
C09172=1111.669,-59.343,-48.752,179.747,5.346,149.007
C09173=1111.673,-59.558,-48.742,179.747,5.343,149.006
C09174=1111.678,-59.772,-48.732,179.746,5.338,149.005
C09175=1111.682,-59.987,-48.722,179.746,5.334,149.004
C09176=1111.687,-60.237,-48.711,179.747,5.329,149.003
C09177=1111.692,-60.487,-48.699,179.746,5.324,149.002
C09178=1111.697,-60.736,-48.688,179.746,5.319,149.001
C09179=1111.703,-60.986,-48.676,179.745,5.314,149.000
C09180=1111.708,-61.236,-48.666,179.744,5.309,148.999
C09181=1111.713,-61.486,-48.654,179.744,5.304,148.998
C09182=1111.718,-61.735,-48.643,179.743,5.298,148.997
C09183=1111.724,-61.985,-48.631,179.743,5.293,148.996
C09184=1111.729,-62.234,-48.620,179.743,5.289,148.995
C09185=1111.734,-62.484,-48.608,179.743,5.284,148.994
C09186=1111.739,-62.734,-48.597,179.742,5.279,148.993
C09187=1111.744,-62.984,-48.586,179.741,5.273,148.992
C09188=1111.750,-63.233,-48.574,179.742,5.268,148.991
C09189=1111.755,-63.483,-48.563,179.741,5.263,148.990
C09190=1111.760,-63.733,-48.551,179.741,5.259,148.989
C09191=1111.765,-63.982,-48.540,179.740,5.253,148.988
C09192=1111.770,-64.232,-48.530,179.740,5.248,148.987
C09193=1111.776,-64.482,-48.518,179.740,5.243,148.986
C09194=1111.780,-64.732,-48.507,179.740,5.238,148.985
C09195=1111.787,-64.981,-48.495,179.739,5.232,148.984
C09196=1111.791,-65.230,-48.484,179.739,5.227,148.983
C09197=1111.796,-65.481,-48.473,179.739,5.222,148.982
C09198=1111.802,-65.731,-48.461,179.739,5.217,148.981
